RoboDK station: Estación_kuka_ibero.rdk

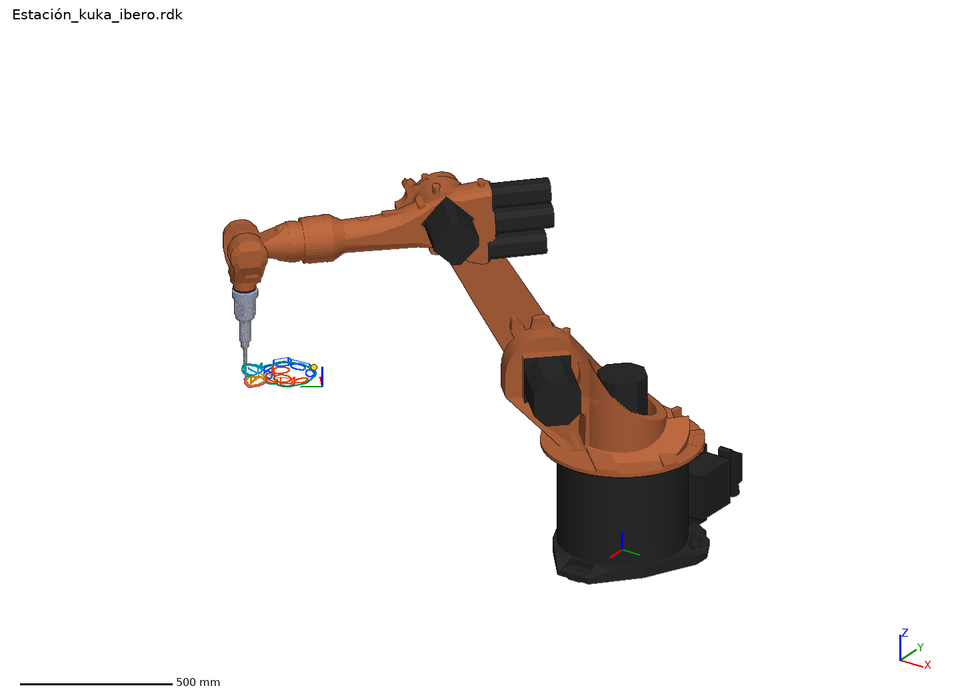
[picture v0: the station drawn from its stored meshes, robots at their saved joint values, targets as dots, program paths as lines]
Station Estación_kuka_ibero (saved by RoboDK 5.9.0). Poses are relative to the parent item; angles as X-Y-Z fixed-axis rotations.
  - frame KUKA KR 16 2 Base at (0, 0, 1020) mm, rotated rx 0 ry 0 rz -90 deg
    - robot KUKA KR 16 2: 6 axes, payload 16 kg, reach 1611 mm, repeatability 0.05 mm, weight 235 kg
        modified DH rows (alpha deg, a mm, theta deg, d mm): 0, 0, 0, 675; -90, 260, 0, 0; 0, 680, -90, 0; -90, -35, 0, 670; 90, 0, 0, 0; -90, 0, 180, 158
        joint limits [-185, -155, -130, -350, -130, -350] to [185, 35, 154, 350, 130, 350]; home [0, -90, 90, 0, 0, 0]; saved at [45.036, -60.88, 62.472, -0.86, 88.364, 45.057]
      - tool Plumon_ensamble, TCP at (4.25, 1.36, 301.29) mm, size 85.6 x 85.6 x 301.8 mm, geometry from Plumon_ensamble.IGS
  - object Celda_completa at (0, 0, 0) mm, size 7080 x 5029 x 2401 mm, geometry from Celda_completa.IGS
  - frame Frame 2 at (-643.65, -798.86, 1757.58) mm, rotated rx -0.03 ry 0.86 rz 129.82 deg
    - object RASPBERRY PI logo-0 at (0, 0, 0) mm
  - machining project P_in_1: rotZ(0) | rotX(0)*rotY(0) | rotz(0) | onStart | onPathStart | onApproach | onPoint | onRetract | onFinish | SetRPM(%1) | SetTool(%1) | Extruder(%1) | default | default | OutOnMov(%1) | OutOffMov(%1) | onPathFinish | M_RunCode(%1) | ag
  - program P_in_1 (855 instructions, listed below)
  - machining project P_in_2: rotZ(0) | rotX(0)*rotY(0) | rotz(0) | onStart | onPathStart | onApproach | onPoint | onRetract | onFinish | SetRPM(%1) | SetTool(%1) | Extruder(%1) | default | default | OutOnMov(%1) | OutOffMov(%1) | onPathFinish | M_RunCode(%1)
  - program P_in_2 (723 instructions, listed below)
  - machining project P_ou_1: rotZ(0) | rotX(0)*rotY(0) | rotz(0) | onStart | onPathStart | onApproach | onPoint | onRetract | onFinish | SetRPM(%1) | SetTool(%1) | Extruder(%1) | default | default | OutOnMov(%1) | OutOffMov(%1) | onPathFinish | M_RunCode(%1)
  - program P_ou_1 (860 instructions, listed below)
  - machining project P_ou_2: rotZ(0) | rotX(0)*rotY(0) | rotz(0) | onStart | onPathStart | onApproach | onPoint | onRetract | onFinish | SetRPM(%1) | SetTool(%1) | Extruder(%1) | default | default | OutOnMov(%1) | OutOffMov(%1) | onPathFinish | M_RunCode(%1)
  - program P_ou_2 (404 instructions, listed below)
  - machining project P_fl_1: rotZ(0) | rotX(0)*rotY(0) | rotz(0) | onStart | onPathStart | onApproach | onPoint | onRetract | onFinish | SetRPM(%1) | SetTool(%1) | Extruder(%1) | default | default | OutOnMov(%1) | OutOffMov(%1) | onPathFinish | M_RunCode(%1)
  - program P_fl_1 (618 instructions, listed below)
  - machining project P_fl_2: rotZ(0) | rotX(0)*rotY(0) | rotz(0) | onStart | onPathStart | onApproach | onPoint | onRetract | onFinish | SetRPM(%1) | SetTool(%1) | Extruder(%1) | default | default | OutOnMov(%1) | OutOffMov(%1) | onPathFinish | M_RunCode(%1)
  - program P_fl_2 (611 instructions, listed below)
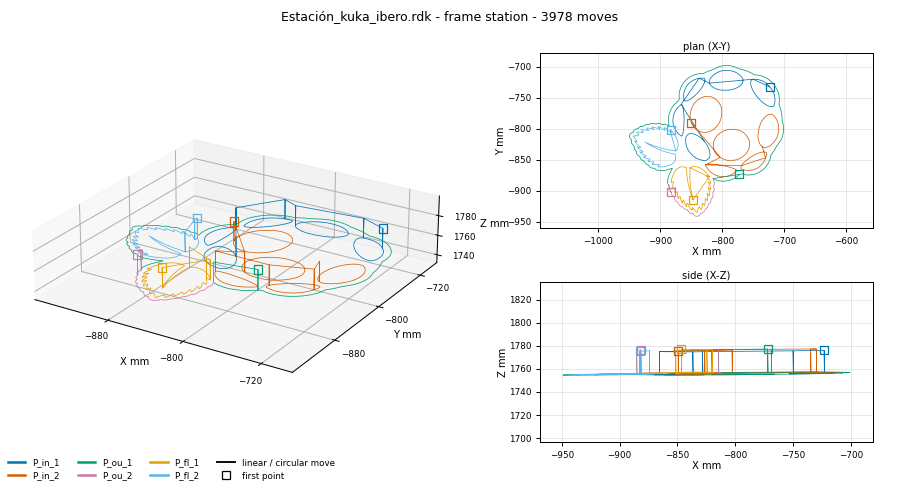
[picture p0: tool path of Estación_kuka_ibero.rdk in frame station, 3978 of 3978 moves have a stored position in this frame; points joined in program order, loops and branches not executed]

--- program P_in_1 (robot KUKA KR 16 2) ---
  Suave(1)
  Establecer velocidad (1000.0 mm/s)
  Est. Ref.: Frame 2
  Est. herr: Plumon_ensamble
  Mostrar Plumon_ensamble
  MoveJ 1 to (101.69, 18.24, 20) mm, rotated rx -180 ry 0 rz -39.83 deg; joints [44.906, -80.315, 88.498, -0.868, 81.773, 45.027]
  MoveL 2 to (101.69, 18.24, 20) mm, rotated rx -180 ry 0 rz -39.83 deg; joints [44.906, -80.315, 88.498, -0.868, 81.773, 45.027]
  MoveL 3 to (101.69, 18.24, 0) mm, rotated rx 180 ry 0 rz -39.83 deg; joints [44.889, -79.963, 89.829, -0.872, 80.089, 45.036]
  MoveL 4 to (101.69, 18.24, 0) mm, rotated rx 180 ry 0 rz -39.83 deg; joints [44.889, -79.963, 89.829, -0.872, 80.089, 45.036]
  Establecer velocidad (50.0 mm/s)
  MoveL 5 to (102.01, 18.23, 0) mm, rotated rx -180 ry 0 rz -39.83 deg; joints [44.907, -79.966, 89.833, -0.872, 80.088, 45.054]
  MoveL 6 to (102.33, 18.22, 0) mm, rotated rx -180 ry 0 rz -39.83 deg; joints [44.925, -79.969, 89.836, -0.872, 80.088, 45.071]
  MoveL 7 to (102.65, 18.22, 0) mm, rotated rx 180 ry 0 rz -39.83 deg; joints [44.942, -79.971, 89.84, -0.872, 80.087, 45.089]
  MoveL 8 to (102.97, 18.21, 0) mm, rotated rx 180 ry 0 rz -39.83 deg; joints [44.96, -79.974, 89.844, -0.872, 80.086, 45.106]
  MoveL 9 to (103.82, 18.21, 0) mm, rotated rx 180 ry 0 rz -39.83 deg; joints [45.007, -79.981, 89.853, -0.873, 80.085, 45.153]
  MoveL 10 to (104.66, 18.21, 0) mm, rotated rx 180 ry 0 rz -39.83 deg; joints [45.053, -79.986, 89.86, -0.873, 80.083, 45.2]
  MoveL 11 to (105.51, 18.24, 0) mm, rotated rx -180 ry 0 rz -39.83 deg; joints [45.1, -79.99, 89.866, -0.873, 80.082, 45.247]
  MoveL 12 to (106.35, 18.29, 0) mm, rotated rx 180 ry 0 rz -39.83 deg; joints [45.147, -79.991, 89.869, -0.873, 80.081, 45.294]
  MoveL 13 to (107.28, 18.4, 0) mm, rotated rx 180 ry 0 rz -39.83 deg; joints [45.199, -79.989, 89.867, -0.873, 80.081, 45.346]
  MoveL 14 to (108.21, 18.54, 0) mm, rotated rx 180 ry 0 rz -39.83 deg; joints [45.251, -79.984, 89.863, -0.873, 80.082, 45.398]
  MoveL 15 to (109.14, 18.7, 0) mm, rotated rx 180 ry 0 rz -39.83 deg; joints [45.303, -79.977, 89.855, -0.873, 80.083, 45.45]
  MoveL 16 to (110.07, 18.89, 0) mm, rotated rx 180 ry 0 rz -39.83 deg; joints [45.355, -79.968, 89.846, -0.873, 80.084, 45.502]
  MoveL 17 to (110.67, 19.01, 0) mm, rotated rx 180 ry 0 rz -39.83 deg; joints [45.389, -79.961, 89.839, -0.873, 80.085, 45.536]
  MoveL 18 to (111.27, 19.15, 0) mm, rotated rx -180 ry 0 rz -39.83 deg; joints [45.423, -79.954, 89.831, -0.873, 80.086, 45.57]
  MoveL 19 to (111.86, 19.3, 0) mm, rotated rx 180 ry 0 rz -39.83 deg; joints [45.456, -79.946, 89.822, -0.873, 80.087, 45.603]
  MoveL 20 to (112.45, 19.46, 0) mm, rotated rx 180 ry 0 rz -39.83 deg; joints [45.49, -79.936, 89.811, -0.873, 80.089, 45.636]
  MoveL 21 to (112.98, 19.63, 0) mm, rotated rx 180 ry 0 rz -39.83 deg; joints [45.52, -79.926, 89.8, -0.873, 80.09, 45.666]
  MoveL 22 to (113.5, 19.82, 0) mm, rotated rx -180 ry 0 rz -39.83 deg; joints [45.549, -79.914, 89.786, -0.873, 80.092, 45.696]
  MoveL 23 to (114.02, 20.01, 0) mm, rotated rx 180 ry 0 rz -39.83 deg; joints [45.579, -79.901, 89.772, -0.873, 80.094, 45.726]
  MoveL 24 to (114.54, 20.22, 0) mm, rotated rx -180 ry 0 rz -39.83 deg; joints [45.608, -79.888, 89.757, -0.873, 80.096, 45.755]
  MoveL 25 to (114.92, 20.37, 0) mm, rotated rx -180 ry 0 rz -39.83 deg; joints [45.63, -79.877, 89.745, -0.873, 80.098, 45.777]
  MoveL 26 to (115.3, 20.53, 0) mm, rotated rx 180 ry 0 rz -39.83 deg; joints [45.652, -79.867, 89.733, -0.873, 80.1, 45.799]
  MoveL 27 to (115.68, 20.69, 0) mm, rotated rx 180 ry 0 rz -39.83 deg; joints [45.674, -79.856, 89.721, -0.873, 80.102, 45.82]
  MoveL 28 to (116.05, 20.86, 0) mm, rotated rx 180 ry 0 rz -39.83 deg; joints [45.695, -79.844, 89.707, -0.873, 80.104, 45.842]
  MoveL 29 to (116.62, 21.14, 0) mm, rotated rx -180 ry 0 rz -39.83 deg; joints [45.728, -79.825, 89.686, -0.873, 80.107, 45.874]
  MoveL 30 to (117.19, 21.42, 0) mm, rotated rx -180 ry 0 rz -39.83 deg; joints [45.76, -79.805, 89.663, -0.873, 80.11, 45.907]
  MoveL 31 to (117.75, 21.72, 0) mm, rotated rx -180 ry 0 rz -39.83 deg; joints [45.792, -79.784, 89.638, -0.873, 80.114, 45.939]
  MoveL 32 to (118.3, 22.03, 0) mm, rotated rx -180 ry 0 rz -39.83 deg; joints [45.824, -79.762, 89.613, -0.873, 80.118, 45.97]
  MoveL 33 to (118.89, 22.38, 0) mm, rotated rx 180 ry 0 rz -39.83 deg; joints [45.858, -79.737, 89.584, -0.873, 80.122, 46.004]
  MoveL 34 to (119.47, 22.73, 0) mm, rotated rx -180 ry 0 rz -39.83 deg; joints [45.892, -79.712, 89.555, -0.873, 80.126, 46.038]
  MoveL 35 to (120.05, 23.09, 0) mm, rotated rx -180 ry 0 rz -39.83 deg; joints [45.925, -79.685, 89.525, -0.873, 80.131, 46.071]
  MoveL 36 to (120.62, 23.46, 0) mm, rotated rx 180 ry 0 rz -39.83 deg; joints [45.958, -79.658, 89.493, -0.873, 80.136, 46.104]
  MoveL 37 to (121.16, 23.83, 0) mm, rotated rx -180 ry 0 rz -39.83 deg; joints [45.989, -79.631, 89.462, -0.873, 80.141, 46.135]
  MoveL 38 to (121.69, 24.21, 0) mm, rotated rx 180 ry 0 rz -39.83 deg; joints [46.02, -79.603, 89.429, -0.873, 80.146, 46.166]
  MoveL 39 to (122.22, 24.59, 0) mm, rotated rx -180 ry 0 rz -39.83 deg; joints [46.05, -79.574, 89.396, -0.873, 80.151, 46.196]
  MoveL 40 to (122.73, 24.99, 0) mm, rotated rx 180 ry 0 rz -39.83 deg; joints [46.08, -79.545, 89.361, -0.873, 80.156, 46.226]
  MoveL 41 to (123.24, 25.41, 0) mm, rotated rx 180 ry 0 rz -39.83 deg; joints [46.11, -79.513, 89.325, -0.873, 80.162, 46.256]
  MoveL 42 to (123.74, 25.84, 0) mm, rotated rx 180 ry 0 rz -39.83 deg; joints [46.139, -79.481, 89.287, -0.873, 80.168, 46.285]
  MoveL 43 to (124.23, 26.28, 0) mm, rotated rx 180 ry 0 rz -39.83 deg; joints [46.168, -79.447, 89.247, -0.873, 80.174, 46.313]
  MoveL 44 to (124.7, 26.74, 0) mm, rotated rx -180 ry 0 rz -39.83 deg; joints [46.195, -79.412, 89.206, -0.873, 80.18, 46.341]
  MoveL 45 to (125.16, 27.22, 0) mm, rotated rx 180 ry 0 rz -39.83 deg; joints [46.223, -79.375, 89.163, -0.873, 80.187, 46.368]
  MoveL 46 to (125.61, 27.71, 0) mm, rotated rx 180 ry 0 rz -39.83 deg; joints [46.249, -79.337, 89.118, -0.873, 80.194, 46.394]
  MoveL 47 to (126.06, 28.2, 0) mm, rotated rx 180 ry 0 rz -39.83 deg; joints [46.276, -79.299, 89.074, -0.873, 80.201, 46.421]
  MoveL 48 to (126.51, 28.69, 0) mm, rotated rx 180 ry 0 rz -39.83 deg; joints [46.302, -79.262, 89.03, -0.873, 80.208, 46.448]
  MoveL 49 to (126.76, 28.95, 0) mm, rotated rx 180 ry 0 rz -39.83 deg; joints [46.317, -79.242, 89.006, -0.873, 80.212, 46.462]
  MoveL 50 to (127.01, 29.21, 0) mm, rotated rx 180 ry 0 rz -39.83 deg; joints [46.332, -79.222, 88.983, -0.873, 80.216, 46.477]
  MoveL 51 to (127.25, 29.47, 0) mm, rotated rx 180 ry 0 rz -39.83 deg; joints [46.346, -79.202, 88.959, -0.873, 80.22, 46.491]
  MoveL 52 to (127.48, 29.74, 0) mm, rotated rx -180 ry 0 rz -39.83 deg; joints [46.36, -79.18, 88.934, -0.873, 80.224, 46.504]
  MoveL 53 to (127.71, 30.06, 0) mm, rotated rx 180 ry 0 rz -39.83 deg; joints [46.373, -79.156, 88.905, -0.873, 80.228, 46.518]
  MoveL 54 to (127.92, 30.38, 0) mm, rotated rx -180 ry 0 rz -39.83 deg; joints [46.386, -79.131, 88.874, -0.873, 80.233, 46.531]
  MoveL 55 to (128.12, 30.71, 0) mm, rotated rx 180 ry 0 rz -39.83 deg; joints [46.398, -79.104, 88.843, -0.873, 80.238, 46.543]
  MoveL 56 to (128.32, 31.05, 0) mm, rotated rx 180 ry 0 rz -39.83 deg; joints [46.41, -79.077, 88.812, -0.873, 80.243, 46.555]
  Establecer velocidad (1000.0 mm/s)
  MoveL 57 to (128.32, 31.05, 0) mm, rotated rx 180 ry 0 rz -39.83 deg; joints [46.41, -79.077, 88.812, -0.873, 80.243, 46.555]
  MoveL 58 to (128.32, 31.05, 20) mm, rotated rx 180 ry 0 rz -39.83 deg; joints [46.427, -79.425, 87.481, -0.869, 81.922, 46.545]
  Establecer velocidad (1000.0 mm/s)
  MoveL 59 to (101.69, 18.24, 20) mm, rotated rx -180 ry 0 rz -39.83 deg; joints [44.906, -80.315, 88.498, -0.868, 81.773, 45.027]
  MoveL 60 to (101.69, 18.24, 0) mm, rotated rx 180 ry 0 rz -39.83 deg; joints [44.889, -79.963, 89.829, -0.872, 80.089, 45.036]
  MoveL 61 to (101.69, 18.24, 0) mm, rotated rx 180 ry 0 rz -39.83 deg; joints [44.889, -79.963, 89.829, -0.872, 80.089, 45.036]
  Establecer velocidad (50.0 mm/s)
  MoveL 62 to (101.37, 18.23, 0) mm, rotated rx -180 ry 0 rz -39.83 deg; joints [44.872, -79.961, 89.826, -0.872, 80.089, 45.018]
  MoveL 63 to (101.06, 18.22, 0) mm, rotated rx 180 ry 0 rz -39.83 deg; joints [44.854, -79.959, 89.824, -0.872, 80.09, 45.001]
  MoveL 64 to (100.74, 18.22, 0) mm, rotated rx 180 ry 0 rz -39.83 deg; joints [44.836, -79.957, 89.821, -0.872, 80.09, 44.983]
  MoveL 65 to (100.42, 18.21, 0) mm, rotated rx 180 ry 0 rz -39.83 deg; joints [44.819, -79.955, 89.818, -0.872, 80.091, 44.965]
  MoveL 66 to (99.57, 18.21, 0) mm, rotated rx -180 ry 0 rz -39.83 deg; joints [44.772, -79.95, 89.811, -0.872, 80.092, 44.918]
  MoveL 67 to (98.72, 18.21, 0) mm, rotated rx 180 ry 0 rz -39.83 deg; joints [44.725, -79.943, 89.801, -0.872, 80.094, 44.872]
  MoveL 68 to (97.88, 18.24, 0) mm, rotated rx 180 ry 0 rz -39.83 deg; joints [44.679, -79.935, 89.79, -0.872, 80.096, 44.825]
  MoveL 69 to (97.04, 18.29, 0) mm, rotated rx 180 ry 0 rz -39.83 deg; joints [44.633, -79.924, 89.776, -0.872, 80.098, 44.779]
  MoveL 70 to (96.1, 18.4, 0) mm, rotated rx 180 ry 0 rz -39.83 deg; joints [44.582, -79.908, 89.756, -0.872, 80.102, 44.728]
  MoveL 71 to (95.17, 18.54, 0) mm, rotated rx 180 ry 0 rz -39.83 deg; joints [44.531, -79.889, 89.733, -0.872, 80.105, 44.677]
  MoveL 72 to (94.25, 18.7, 0) mm, rotated rx 180 ry 0 rz -39.83 deg; joints [44.481, -79.868, 89.707, -0.872, 80.11, 44.627]
  MoveL 73 to (93.32, 18.89, 0) mm, rotated rx 180 ry 0 rz -39.83 deg; joints [44.431, -79.846, 89.679, -0.872, 80.114, 44.577]
  MoveL 74 to (92.72, 19.01, 0) mm, rotated rx -180 ry 0 rz -39.83 deg; joints [44.398, -79.831, 89.661, -0.872, 80.117, 44.544]
  MoveL 75 to (92.12, 19.15, 0) mm, rotated rx 180 ry 0 rz -39.83 deg; joints [44.366, -79.815, 89.641, -0.872, 80.121, 44.512]
  MoveL 76 to (91.53, 19.3, 0) mm, rotated rx 180 ry 0 rz -39.83 deg; joints [44.334, -79.798, 89.62, -0.872, 80.124, 44.48]
  MoveL 77 to (90.94, 19.46, 0) mm, rotated rx 180 ry 0 rz -39.83 deg; joints [44.303, -79.779, 89.598, -0.872, 80.128, 44.449]
  MoveL 78 to (90.41, 19.63, 0) mm, rotated rx 180 ry 0 rz -39.83 deg; joints [44.275, -79.761, 89.576, -0.872, 80.131, 44.42]
  MoveL 79 to (89.89, 19.82, 0) mm, rotated rx -180 ry 0 rz -39.83 deg; joints [44.247, -79.742, 89.552, -0.872, 80.135, 44.393]
  MoveL 80 to (89.37, 20.01, 0) mm, rotated rx 180 ry 0 rz -39.83 deg; joints [44.219, -79.722, 89.527, -0.872, 80.139, 44.365]
  MoveL 81 to (88.85, 20.22, 0) mm, rotated rx 180 ry 0 rz -39.83 deg; joints [44.192, -79.701, 89.502, -0.872, 80.143, 44.338]
  MoveL 82 to (88.47, 20.37, 0) mm, rotated rx 180 ry 0 rz -39.83 deg; joints [44.172, -79.685, 89.482, -0.872, 80.146, 44.318]
  MoveL 83 to (88.09, 20.53, 0) mm, rotated rx 180 ry 0 rz -39.83 deg; joints [44.152, -79.669, 89.463, -0.872, 80.15, 44.297]
  MoveL 84 to (87.71, 20.69, 0) mm, rotated rx 180 ry 0 rz -39.83 deg; joints [44.132, -79.652, 89.443, -0.872, 80.153, 44.278]
  MoveL 85 to (87.33, 20.86, 0) mm, rotated rx -180 ry 0 rz -39.83 deg; joints [44.112, -79.635, 89.422, -0.872, 80.156, 44.258]
  MoveL 86 to (86.76, 21.14, 0) mm, rotated rx 180 ry 0 rz -39.83 deg; joints [44.083, -79.608, 89.389, -0.871, 80.162, 44.228]
  MoveL 87 to (86.2, 21.42, 0) mm, rotated rx 180 ry 0 rz -39.83 deg; joints [44.053, -79.58, 89.355, -0.871, 80.167, 44.199]
  MoveL 88 to (85.64, 21.72, 0) mm, rotated rx 180 ry 0 rz -39.83 deg; joints [44.025, -79.55, 89.319, -0.871, 80.173, 44.17]
  MoveL 89 to (85.09, 22.03, 0) mm, rotated rx -180 ry 0 rz -39.83 deg; joints [43.996, -79.52, 89.283, -0.871, 80.179, 44.141]
  MoveL 90 to (84.5, 22.38, 0) mm, rotated rx 180 ry 0 rz -39.83 deg; joints [43.966, -79.487, 89.242, -0.871, 80.186, 44.111]
  MoveL 91 to (83.91, 22.73, 0) mm, rotated rx 180 ry 0 rz -39.83 deg; joints [43.936, -79.453, 89.201, -0.871, 80.192, 44.081]
  MoveL 92 to (83.34, 23.09, 0) mm, rotated rx 180 ry 0 rz -39.83 deg; joints [43.906, -79.419, 89.16, -0.871, 80.199, 44.051]
  MoveL 93 to (82.76, 23.46, 0) mm, rotated rx -180 ry 0 rz -39.83 deg; joints [43.877, -79.383, 89.117, -0.871, 80.206, 44.022]
  MoveL 94 to (82.23, 23.83, 0) mm, rotated rx 180 ry 0 rz -39.83 deg; joints [43.85, -79.349, 89.075, -0.871, 80.213, 43.994]
  MoveL 95 to (81.7, 24.21, 0) mm, rotated rx 180 ry 0 rz -39.83 deg; joints [43.823, -79.313, 89.032, -0.871, 80.22, 43.967]
  MoveL 96 to (81.17, 24.59, 0) mm, rotated rx 180 ry 0 rz -39.83 deg; joints [43.797, -79.277, 88.988, -0.871, 80.228, 43.941]
  MoveL 97 to (80.66, 24.99, 0) mm, rotated rx 180 ry 0 rz -39.83 deg; joints [43.771, -79.24, 88.943, -0.871, 80.235, 43.915]
  MoveL 98 to (80.15, 25.41, 0) mm, rotated rx 180 ry 0 rz -39.83 deg; joints [43.746, -79.201, 88.896, -0.871, 80.243, 43.89]
  MoveL 99 to (79.65, 25.84, 0) mm, rotated rx 180 ry 0 rz -39.83 deg; joints [43.721, -79.162, 88.848, -0.871, 80.251, 43.865]
  MoveL 100 to (79.16, 26.28, 0) mm, rotated rx 180 ry 0 rz -39.83 deg; joints [43.697, -79.121, 88.799, -0.871, 80.259, 43.841]
  MoveL 101 to (78.69, 26.74, 0) mm, rotated rx 180 ry 0 rz -39.83 deg; joints [43.675, -79.079, 88.748, -0.871, 80.267, 43.818]
  MoveL 102 to (78.23, 27.22, 0) mm, rotated rx -180 ry 0 rz -39.83 deg; joints [43.653, -79.036, 88.696, -0.871, 80.276, 43.796]
  MoveL 103 to (77.78, 27.71, 0) mm, rotated rx 180 ry 0 rz -39.83 deg; joints [43.631, -78.992, 88.642, -0.871, 80.285, 43.774]
  MoveL 104 to (77.33, 28.2, 0) mm, rotated rx -180 ry 0 rz -39.83 deg; joints [43.61, -78.947, 88.589, -0.871, 80.294, 43.753]
  MoveL 105 to (76.88, 28.69, 0) mm, rotated rx -180 ry 0 rz -39.83 deg; joints [43.588, -78.904, 88.535, -0.871, 80.303, 43.731]
  MoveL 106 to (76.63, 28.95, 0) mm, rotated rx -180 ry 0 rz -39.83 deg; joints [43.576, -78.88, 88.507, -0.871, 80.308, 43.719]
  MoveL 107 to (76.38, 29.21, 0) mm, rotated rx 180 ry 0 rz -39.83 deg; joints [43.564, -78.857, 88.479, -0.87, 80.313, 43.707]
  MoveL 108 to (76.14, 29.47, 0) mm, rotated rx 180 ry 0 rz -39.83 deg; joints [43.553, -78.833, 88.45, -0.87, 80.318, 43.695]
  MoveL 109 to (75.91, 29.74, 0) mm, rotated rx 180 ry 0 rz -39.83 deg; joints [43.542, -78.808, 88.42, -0.87, 80.323, 43.684]
  MoveL 110 to (75.68, 30.06, 0) mm, rotated rx 180 ry 0 rz -39.83 deg; joints [43.531, -78.781, 88.387, -0.87, 80.329, 43.674]
  MoveL 111 to (75.47, 30.38, 0) mm, rotated rx 180 ry 0 rz -39.83 deg; joints [43.522, -78.752, 88.352, -0.87, 80.335, 43.664]
  MoveL 112 to (75.27, 30.71, 0) mm, rotated rx -180 ry 0 rz -39.83 deg; joints [43.513, -78.723, 88.317, -0.87, 80.341, 43.656]
  MoveL 113 to (75.07, 31.05, 0) mm, rotated rx 180 ry 0 rz -39.83 deg; joints [43.505, -78.694, 88.281, -0.87, 80.347, 43.647]
  MoveL 114 to (75.07, 31.05, 0) mm, rotated rx 180 ry 0 rz -39.83 deg; joints [43.505, -78.694, 88.281, -0.87, 80.347, 43.647]
  MoveL 115 to (74.94, 31.32, 0) mm, rotated rx -180 ry 0 rz -39.83 deg; joints [43.5, -78.671, 88.253, -0.87, 80.351, 43.642]
  MoveL 116 to (74.82, 31.59, 0) mm, rotated rx 180 ry 0 rz -39.83 deg; joints [43.495, -78.648, 88.225, -0.87, 80.356, 43.637]
  MoveL 117 to (74.7, 31.86, 0) mm, rotated rx 180 ry 0 rz -39.83 deg; joints [43.49, -78.624, 88.197, -0.87, 80.361, 43.632]
  MoveL 118 to (74.6, 32.14, 0) mm, rotated rx 180 ry 0 rz -39.83 deg; joints [43.486, -78.601, 88.168, -0.87, 80.366, 43.628]
  MoveL 119 to (74.52, 32.35, 0) mm, rotated rx -180 ry 0 rz -39.83 deg; joints [43.483, -78.583, 88.147, -0.87, 80.37, 43.625]
  MoveL 120 to (74.46, 32.56, 0) mm, rotated rx 180 ry 0 rz -39.83 deg; joints [43.481, -78.565, 88.125, -0.87, 80.373, 43.623]
  MoveL 121 to (74.41, 32.78, 0) mm, rotated rx 180 ry 0 rz -39.83 deg; joints [43.48, -78.547, 88.103, -0.87, 80.377, 43.622]
  MoveL 122 to (74.37, 33, 0) mm, rotated rx 180 ry 0 rz -39.83 deg; joints [43.479, -78.528, 88.081, -0.87, 80.381, 43.621]
  MoveL 123 to (74.33, 33.36, 0) mm, rotated rx 180 ry 0 rz -39.83 deg; joints [43.479, -78.498, 88.045, -0.87, 80.387, 43.621]
  MoveL 124 to (74.32, 33.72, 0) mm, rotated rx 180 ry 0 rz -39.83 deg; joints [43.481, -78.469, 88.009, -0.87, 80.393, 43.622]
  MoveL 125 to (74.35, 34.09, 0) mm, rotated rx 180 ry 0 rz -39.83 deg; joints [43.485, -78.439, 87.973, -0.87, 80.4, 43.626]
  MoveL 126 to (74.42, 34.44, 0) mm, rotated rx 180 ry 0 rz -39.83 deg; joints [43.491, -78.411, 87.939, -0.87, 80.405, 43.632]
  MoveL 127 to (74.51, 34.76, 0) mm, rotated rx 180 ry 0 rz -39.83 deg; joints [43.498, -78.386, 87.909, -0.87, 80.411, 43.639]
  MoveL 128 to (74.63, 35.07, 0) mm, rotated rx 180 ry 0 rz -39.83 deg; joints [43.506, -78.362, 87.88, -0.87, 80.416, 43.647]
  MoveL 129 to (74.77, 35.37, 0) mm, rotated rx 180 ry 0 rz -39.83 deg; joints [43.516, -78.338, 87.852, -0.87, 80.42, 43.657]
  MoveL 130 to (74.94, 35.65, 0) mm, rotated rx 180 ry 0 rz -39.83 deg; joints [43.527, -78.316, 87.826, -0.87, 80.425, 43.668]
  MoveL 131 to (75.22, 36.07, 0) mm, rotated rx 180 ry 0 rz -39.83 deg; joints [43.544, -78.285, 87.788, -0.87, 80.432, 43.685]
  MoveL 132 to (75.53, 36.47, 0) mm, rotated rx 180 ry 0 rz -39.83 deg; joints [43.564, -78.255, 87.752, -0.87, 80.438, 43.705]
  MoveL 133 to (75.87, 36.85, 0) mm, rotated rx 180 ry 0 rz -39.83 deg; joints [43.584, -78.228, 87.719, -0.87, 80.443, 43.725]
  MoveL 134 to (76.23, 37.2, 0) mm, rotated rx -180 ry 0 rz -39.83 deg; joints [43.606, -78.202, 87.689, -0.87, 80.449, 43.747]
  MoveL 135 to (76.54, 37.48, 0) mm, rotated rx -180 ry 0 rz -39.83 deg; joints [43.624, -78.182, 87.665, -0.87, 80.453, 43.765]
  MoveL 136 to (76.85, 37.75, 0) mm, rotated rx 180 ry 0 rz -39.83 deg; joints [43.643, -78.163, 87.643, -0.87, 80.457, 43.784]
  MoveL 137 to (77.18, 38.01, 0) mm, rotated rx 180 ry 0 rz -39.83 deg; joints [43.662, -78.145, 87.621, -0.87, 80.46, 43.803]
  MoveL 138 to (77.51, 38.26, 0) mm, rotated rx 180 ry 0 rz -39.83 deg; joints [43.682, -78.127, 87.6, -0.87, 80.464, 43.822]
  MoveL 139 to (78.01, 38.62, 0) mm, rotated rx 180 ry 0 rz -39.83 deg; joints [43.711, -78.102, 87.57, -0.87, 80.469, 43.851]
  MoveL 140 to (78.52, 38.97, 0) mm, rotated rx 180 ry 0 rz -39.83 deg; joints [43.741, -78.078, 87.542, -0.87, 80.474, 43.881]
  MoveL 141 to (79.04, 39.3, 0) mm, rotated rx 180 ry 0 rz -39.83 deg; joints [43.77, -78.056, 87.515, -0.87, 80.478, 43.911]
  MoveL 142 to (79.57, 39.61, 0) mm, rotated rx 180 ry 0 rz -39.83 deg; joints [43.801, -78.035, 87.491, -0.87, 80.483, 43.941]
  MoveL 143 to (80.13, 39.9, 0) mm, rotated rx 180 ry 0 rz -39.83 deg; joints [43.833, -78.016, 87.469, -0.87, 80.486, 43.973]
  MoveL 144 to (80.71, 40.17, 0) mm, rotated rx 180 ry 0 rz -39.83 deg; joints [43.866, -77.999, 87.449, -0.87, 80.49, 44.006]
  MoveL 145 to (81.29, 40.42, 0) mm, rotated rx 180 ry 0 rz -39.83 deg; joints [43.899, -77.984, 87.431, -0.87, 80.493, 44.039]
  MoveL 146 to (81.88, 40.66, 0) mm, rotated rx -180 ry 0 rz -39.83 deg; joints [43.932, -77.969, 87.414, -0.87, 80.496, 44.072]
  MoveL 147 to (82.65, 40.97, 0) mm, rotated rx 180 ry 0 rz -39.83 deg; joints [43.975, -77.951, 87.392, -0.87, 80.499, 44.115]
  MoveL 148 to (83.42, 41.27, 0) mm, rotated rx -180 ry 0 rz -39.83 deg; joints [44.018, -77.933, 87.372, -0.871, 80.503, 44.158]
  MoveL 149 to (84.2, 41.55, 0) mm, rotated rx 180 ry 0 rz -39.83 deg; joints [44.062, -77.916, 87.353, -0.871, 80.506, 44.202]
  MoveL 150 to (84.98, 41.81, 0) mm, rotated rx 180 ry 0 rz -39.83 deg; joints [44.106, -77.902, 87.336, -0.871, 80.509, 44.246]
  MoveL 151 to (86.19, 42.17, 0) mm, rotated rx 180 ry 0 rz -39.83 deg; joints [44.173, -77.882, 87.314, -0.871, 80.512, 44.312]
  MoveL 152 to (87.4, 42.48, 0) mm, rotated rx 180 ry 0 rz -39.83 deg; joints [44.24, -77.867, 87.296, -0.871, 80.515, 44.38]
  MoveL 153 to (88.63, 42.76, 0) mm, rotated rx 180 ry 0 rz -39.83 deg; joints [44.307, -77.854, 87.283, -0.871, 80.517, 44.447]
  MoveL 154 to (89.86, 43.01, 0) mm, rotated rx -180 ry 0 rz -39.83 deg; joints [44.375, -77.844, 87.272, -0.871, 80.519, 44.515]
  MoveL 155 to (90.97, 43.22, 0) mm, rotated rx 180 ry 0 rz -39.83 deg; joints [44.436, -77.836, 87.263, -0.871, 80.52, 44.576]
  MoveL 156 to (92.08, 43.41, 0) mm, rotated rx 180 ry 0 rz -39.83 deg; joints [44.497, -77.829, 87.256, -0.871, 80.521, 44.637]
  MoveL 157 to (93.2, 43.58, 0) mm, rotated rx 180 ry 0 rz -39.83 deg; joints [44.558, -77.823, 87.251, -0.871, 80.522, 44.698]
  MoveL 158 to (94.31, 43.74, 0) mm, rotated rx 180 ry 0 rz -39.83 deg; joints [44.619, -77.819, 87.248, -0.871, 80.522, 44.759]
  MoveL 159 to (95.45, 43.87, 0) mm, rotated rx 180 ry 0 rz -39.83 deg; joints [44.68, -77.817, 87.246, -0.871, 80.522, 44.82]
  MoveL 160 to (96.62, 43.98, 0) mm, rotated rx 180 ry 0 rz -39.83 deg; joints [44.744, -77.817, 87.247, -0.871, 80.522, 44.884]
  MoveL 161 to (97.86, 44.07, 0) mm, rotated rx -180 ry 0 rz -39.83 deg; joints [44.811, -77.819, 87.252, -0.871, 80.52, 44.951]
  MoveL 162 to (99.2, 44.12, 0) mm, rotated rx 180 ry 0 rz -39.83 deg; joints [44.884, -77.825, 87.261, -0.871, 80.518, 45.024]
  MoveL 163 to (100.08, 44.13, 0) mm, rotated rx 180 ry 0 rz -39.83 deg; joints [44.932, -77.83, 87.269, -0.871, 80.517, 45.072]
  MoveL 164 to (100.89, 44.13, 0) mm, rotated rx 180 ry 0 rz -39.83 deg; joints [44.975, -77.836, 87.277, -0.871, 80.515, 45.115]
  MoveL 165 to (101.47, 44.13, 0) mm, rotated rx 180 ry 0 rz -39.83 deg; joints [45.006, -77.84, 87.283, -0.871, 80.514, 45.146]
  MoveL 166 to (101.69, 44.13, 0) mm, rotated rx 180 ry 0 rz -39.83 deg; joints [45.018, -77.842, 87.285, -0.871, 80.513, 45.159]
  MoveL 167 to (101.69, 44.13, 0) mm, rotated rx 180 ry 0 rz -39.83 deg; joints [45.018, -77.842, 87.285, -0.871, 80.513, 45.159]
  MoveL 168 to (101.92, 44.13, 0) mm, rotated rx 180 ry 0 rz -39.83 deg; joints [45.031, -77.843, 87.287, -0.871, 80.513, 45.171]
  MoveL 169 to (102.5, 44.13, 0) mm, rotated rx 180 ry 0 rz -39.83 deg; joints [45.062, -77.847, 87.293, -0.871, 80.512, 45.202]
  MoveL 170 to (103.3, 44.13, 0) mm, rotated rx -180 ry 0 rz -39.83 deg; joints [45.105, -77.853, 87.301, -0.871, 80.51, 45.245]
  MoveL 171 to (104.19, 44.12, 0) mm, rotated rx 180 ry 0 rz -39.83 deg; joints [45.153, -77.86, 87.311, -0.872, 80.508, 45.293]
  MoveL 172 to (105.53, 44.07, 0) mm, rotated rx -180 ry 0 rz -39.83 deg; joints [45.225, -77.874, 87.329, -0.872, 80.505, 45.365]
  MoveL 173 to (106.77, 43.98, 0) mm, rotated rx 180 ry 0 rz -39.83 deg; joints [45.292, -77.889, 87.349, -0.872, 80.501, 45.432]
  MoveL 174 to (107.94, 43.87, 0) mm, rotated rx 180 ry 0 rz -39.83 deg; joints [45.354, -77.906, 87.371, -0.872, 80.496, 45.495]
  MoveL 175 to (109.08, 43.74, 0) mm, rotated rx 180 ry 0 rz -39.83 deg; joints [45.415, -77.925, 87.395, -0.872, 80.492, 45.555]
  MoveL 176 to (110.19, 43.58, 0) mm, rotated rx 180 ry 0 rz -39.83 deg; joints [45.475, -77.945, 87.421, -0.872, 80.487, 45.615]
  MoveL 177 to (111.31, 43.41, 0) mm, rotated rx 180 ry 0 rz -39.83 deg; joints [45.534, -77.966, 87.449, -0.872, 80.482, 45.675]
  MoveL 178 to (112.42, 43.22, 0) mm, rotated rx 180 ry 0 rz -39.83 deg; joints [45.593, -77.989, 87.478, -0.872, 80.476, 45.734]
  MoveL 179 to (113.53, 43.01, 0) mm, rotated rx 180 ry 0 rz -39.83 deg; joints [45.652, -78.012, 87.508, -0.872, 80.471, 45.793]
  MoveL 180 to (114.76, 42.76, 0) mm, rotated rx -180 ry 0 rz -39.83 deg; joints [45.718, -78.04, 87.544, -0.872, 80.464, 45.859]
  MoveL 181 to (115.98, 42.48, 0) mm, rotated rx 180 ry 0 rz -39.83 deg; joints [45.783, -78.071, 87.582, -0.872, 80.457, 45.924]
  MoveL 182 to (117.2, 42.17, 0) mm, rotated rx 180 ry 0 rz -39.83 deg; joints [45.848, -78.104, 87.624, -0.872, 80.449, 45.989]
  MoveL 183 to (118.4, 41.81, 0) mm, rotated rx 180 ry 0 rz -39.83 deg; joints [45.911, -78.14, 87.669, -0.872, 80.441, 46.053]
  MoveL 184 to (119.19, 41.55, 0) mm, rotated rx -180 ry 0 rz -39.83 deg; joints [45.953, -78.166, 87.702, -0.872, 80.435, 46.094]
  MoveL 185 to (119.97, 41.27, 0) mm, rotated rx -180 ry 0 rz -39.83 deg; joints [45.994, -78.194, 87.737, -0.872, 80.428, 46.135]
  MoveL 186 to (120.74, 40.97, 0) mm, rotated rx -180 ry 0 rz -39.83 deg; joints [46.035, -78.223, 87.773, -0.872, 80.422, 46.176]
  MoveL 187 to (121.51, 40.66, 0) mm, rotated rx -180 ry 0 rz -39.83 deg; joints [46.075, -78.252, 87.81, -0.872, 80.415, 46.217]
  MoveL 188 to (122.1, 40.42, 0) mm, rotated rx 180 ry 0 rz -39.83 deg; joints [46.106, -78.275, 87.838, -0.872, 80.41, 46.248]
  MoveL 189 to (122.68, 40.17, 0) mm, rotated rx 180 ry 0 rz -39.83 deg; joints [46.137, -78.299, 87.868, -0.872, 80.405, 46.279]
  MoveL 190 to (123.26, 39.9, 0) mm, rotated rx 180 ry 0 rz -39.83 deg; joints [46.167, -78.325, 87.899, -0.872, 80.399, 46.309]
  MoveL 191 to (123.82, 39.61, 0) mm, rotated rx 180 ry 0 rz -39.83 deg; joints [46.196, -78.351, 87.932, -0.872, 80.393, 46.339]
  MoveL 192 to (124.35, 39.3, 0) mm, rotated rx 180 ry 0 rz -39.83 deg; joints [46.224, -78.38, 87.967, -0.872, 80.387, 46.366]
  MoveL 193 to (124.87, 38.97, 0) mm, rotated rx 180 ry 0 rz -39.83 deg; joints [46.251, -78.41, 88.004, -0.873, 80.381, 46.393]
  MoveL 194 to (125.38, 38.62, 0) mm, rotated rx -180 ry 0 rz -39.83 deg; joints [46.277, -78.441, 88.043, -0.873, 80.374, 46.42]
  MoveL 195 to (125.88, 38.26, 0) mm, rotated rx 180 ry 0 rz -39.83 deg; joints [46.303, -78.473, 88.083, -0.873, 80.367, 46.446]
  MoveL 196 to (126.21, 38.01, 0) mm, rotated rx 180 ry 0 rz -39.83 deg; joints [46.32, -78.496, 88.11, -0.873, 80.362, 46.463]
  MoveL 197 to (126.53, 37.75, 0) mm, rotated rx 180 ry 0 rz -39.83 deg; joints [46.337, -78.519, 88.138, -0.873, 80.357, 46.48]
  MoveL 198 to (126.85, 37.48, 0) mm, rotated rx 180 ry 0 rz -39.83 deg; joints [46.353, -78.542, 88.167, -0.873, 80.352, 46.496]
  MoveL 199 to (127.16, 37.2, 0) mm, rotated rx 180 ry 0 rz -39.83 deg; joints [46.369, -78.567, 88.197, -0.873, 80.347, 46.512]
  MoveL 200 to (127.52, 36.85, 0) mm, rotated rx 180 ry 0 rz -39.83 deg; joints [46.388, -78.598, 88.235, -0.873, 80.34, 46.531]
  MoveL 201 to (127.86, 36.47, 0) mm, rotated rx 180 ry 0 rz -39.83 deg; joints [46.405, -78.63, 88.274, -0.873, 80.333, 46.548]
  MoveL 202 to (128.17, 36.07, 0) mm, rotated rx 180 ry 0 rz -39.83 deg; joints [46.42, -78.664, 88.316, -0.873, 80.326, 46.564]
  MoveL 203 to (128.45, 35.65, 0) mm, rotated rx 180 ry 0 rz -39.83 deg; joints [46.434, -78.7, 88.359, -0.873, 80.319, 46.577]
  MoveL 204 to (128.62, 35.37, 0) mm, rotated rx 180 ry 0 rz -39.83 deg; joints [46.442, -78.725, 88.389, -0.873, 80.314, 46.585]
  MoveL 205 to (128.76, 35.07, 0) mm, rotated rx 180 ry 0 rz -39.83 deg; joints [46.449, -78.75, 88.42, -0.873, 80.309, 46.592]
  MoveL 206 to (128.88, 34.76, 0) mm, rotated rx 180 ry 0 rz -39.83 deg; joints [46.454, -78.776, 88.451, -0.873, 80.303, 46.598]
  MoveL 207 to (128.97, 34.44, 0) mm, rotated rx -180 ry 0 rz -39.83 deg; joints [46.458, -78.802, 88.483, -0.873, 80.298, 46.602]
  MoveL 208 to (129.04, 34.09, 0) mm, rotated rx 180 ry 0 rz -39.83 deg; joints [46.46, -78.832, 88.519, -0.873, 80.292, 46.604]
  MoveL 209 to (129.07, 33.72, 0) mm, rotated rx 180 ry 0 rz -39.83 deg; joints [46.461, -78.862, 88.554, -0.873, 80.286, 46.605]
  MoveL 210 to (129.06, 33.36, 0) mm, rotated rx 180 ry 0 rz -39.83 deg; joints [46.459, -78.892, 88.59, -0.873, 80.28, 46.603]
  MoveL 211 to (129.02, 33, 0) mm, rotated rx 180 ry 0 rz -39.83 deg; joints [46.456, -78.921, 88.626, -0.873, 80.274, 46.6]
  MoveL 212 to (128.98, 32.78, 0) mm, rotated rx 180 ry 0 rz -39.83 deg; joints [46.453, -78.939, 88.647, -0.873, 80.271, 46.597]
  MoveL 213 to (128.93, 32.56, 0) mm, rotated rx 180 ry 0 rz -39.83 deg; joints [46.449, -78.957, 88.668, -0.873, 80.267, 46.593]
  MoveL 214 to (128.86, 32.35, 0) mm, rotated rx -180 ry 0 rz -39.83 deg; joints [46.445, -78.974, 88.688, -0.873, 80.264, 46.589]
  MoveL 215 to (128.79, 32.14, 0) mm, rotated rx 180 ry 0 rz -39.83 deg; joints [46.44, -78.991, 88.708, -0.873, 80.26, 46.584]
  MoveL 216 to (128.69, 31.86, 0) mm, rotated rx 180 ry 0 rz -39.83 deg; joints [46.433, -79.013, 88.735, -0.873, 80.256, 46.578]
  MoveL 217 to (128.57, 31.59, 0) mm, rotated rx 180 ry 0 rz -39.83 deg; joints [46.426, -79.035, 88.761, -0.873, 80.252, 46.57]
  MoveL 218 to (128.44, 31.32, 0) mm, rotated rx 180 ry 0 rz -39.83 deg; joints [46.418, -79.056, 88.786, -0.873, 80.248, 46.562]
  MoveL 219 to (128.32, 31.05, 0) mm, rotated rx 180 ry 0 rz -39.83 deg; joints [46.41, -79.077, 88.812, -0.873, 80.243, 46.555]
  Establecer velocidad (1000.0 mm/s)
  MoveL 220 to (128.32, 31.05, 0) mm, rotated rx 180 ry 0 rz -39.83 deg; joints [46.41, -79.077, 88.812, -0.873, 80.243, 46.555]
  MoveL 221 to (128.32, 31.05, 20) mm, rotated rx 180 ry 0 rz -39.83 deg; joints [46.427, -79.425, 87.481, -0.869, 81.922, 46.545]
  Establecer velocidad (1000.0 mm/s)
  MoveL 222 to (168.4, 89.11, 20) mm, rotated rx -180 ry 0 rz -39.83 deg; joints [48.709, -74.756, 81.792, -0.867, 82.976, 48.812]
  MoveL 223 to (168.4, 89.11, 0) mm, rotated rx 180 ry 0 rz -39.83 deg; joints [48.694, -74.438, 83.125, -0.871, 81.324, 48.822]
  MoveL 224 to (168.4, 89.11, 0) mm, rotated rx 180 ry 0 rz -39.83 deg; joints [48.694, -74.438, 83.125, -0.871, 81.324, 48.822]
  Establecer velocidad (50.0 mm/s)
  MoveL 225 to (167.87, 89.26, 0) mm, rotated rx -180 ry 0 rz -39.83 deg; joints [48.666, -74.425, 83.108, -0.871, 81.328, 48.794]
  MoveL 226 to (167.33, 89.39, 0) mm, rotated rx -180 ry 0 rz -39.83 deg; joints [48.638, -74.412, 83.092, -0.871, 81.332, 48.766]
  MoveL 227 to (166.79, 89.51, 0) mm, rotated rx 180 ry 0 rz -39.83 deg; joints [48.61, -74.401, 83.077, -0.871, 81.335, 48.738]
  MoveL 228 to (166.25, 89.61, 0) mm, rotated rx -180 ry 0 rz -39.83 deg; joints [48.582, -74.392, 83.065, -0.871, 81.338, 48.71]
  MoveL 229 to (165.14, 89.71, 0) mm, rotated rx 180 ry 0 rz -39.83 deg; joints [48.524, -74.382, 83.05, -0.871, 81.341, 48.652]
  MoveL 230 to (164.01, 89.69, 0) mm, rotated rx 180 ry 0 rz -39.83 deg; joints [48.466, -74.381, 83.047, -0.871, 81.342, 48.594]
  MoveL 231 to (162.89, 89.57, 0) mm, rotated rx 180 ry 0 rz -39.83 deg; joints [48.407, -74.388, 83.055, -0.871, 81.341, 48.535]
  MoveL 232 to (161.78, 89.36, 0) mm, rotated rx 180 ry 0 rz -39.83 deg; joints [48.349, -74.403, 83.073, -0.871, 81.337, 48.477]
  MoveL 233 to (160.86, 89.13, 0) mm, rotated rx 180 ry 0 rz -39.83 deg; joints [48.301, -74.42, 83.093, -0.871, 81.333, 48.429]
  MoveL 234 to (159.97, 88.85, 0) mm, rotated rx -180 ry 0 rz -39.83 deg; joints [48.254, -74.44, 83.118, -0.871, 81.328, 48.382]
  MoveL 235 to (159.09, 88.54, 0) mm, rotated rx -180 ry 0 rz -39.83 deg; joints [48.207, -74.464, 83.147, -0.871, 81.322, 48.336]
  MoveL 236 to (158.21, 88.2, 0) mm, rotated rx 180 ry 0 rz -39.83 deg; joints [48.161, -74.49, 83.179, -0.871, 81.315, 48.29]
  MoveL 237 to (157.52, 87.91, 0) mm, rotated rx 180 ry 0 rz -39.83 deg; joints [48.125, -74.512, 83.206, -0.871, 81.309, 48.253]
  MoveL 238 to (156.84, 87.61, 0) mm, rotated rx 180 ry 0 rz -39.83 deg; joints [48.088, -74.535, 83.235, -0.871, 81.303, 48.217]
  MoveL 239 to (156.15, 87.29, 0) mm, rotated rx -180 ry 0 rz -39.83 deg; joints [48.052, -74.56, 83.265, -0.871, 81.297, 48.181]
  MoveL 240 to (155.48, 86.96, 0) mm, rotated rx -180 ry 0 rz -39.83 deg; joints [48.016, -74.585, 83.296, -0.871, 81.29, 48.145]
  MoveL 241 to (154.69, 86.56, 0) mm, rotated rx -180 ry 0 rz -39.83 deg; joints [47.975, -74.616, 83.335, -0.871, 81.282, 48.103]
  MoveL 242 to (153.92, 86.14, 0) mm, rotated rx 180 ry 0 rz -39.83 deg; joints [47.933, -74.648, 83.375, -0.871, 81.274, 48.062]
  MoveL 243 to (153.16, 85.69, 0) mm, rotated rx -180 ry 0 rz -39.83 deg; joints [47.893, -74.683, 83.418, -0.871, 81.265, 48.022]
  MoveL 244 to (152.41, 85.22, 0) mm, rotated rx 180 ry 0 rz -39.83 deg; joints [47.853, -74.719, 83.464, -0.871, 81.255, 47.982]
  MoveL 245 to (151.64, 84.68, 0) mm, rotated rx 180 ry 0 rz -39.83 deg; joints [47.811, -74.761, 83.516, -0.871, 81.244, 47.941]
  MoveL 246 to (150.88, 84.12, 0) mm, rotated rx 180 ry 0 rz -39.83 deg; joints [47.771, -74.806, 83.572, -0.871, 81.232, 47.9]
  MoveL 247 to (150.15, 83.52, 0) mm, rotated rx 180 ry 0 rz -39.83 deg; joints [47.731, -74.853, 83.63, -0.871, 81.22, 47.86]
  MoveL 248 to (149.43, 82.9, 0) mm, rotated rx -180 ry 0 rz -39.83 deg; joints [47.692, -74.901, 83.691, -0.871, 81.207, 47.822]
  MoveL 249 to (148.81, 82.34, 0) mm, rotated rx -180 ry 0 rz -39.83 deg; joints [47.658, -74.946, 83.746, -0.871, 81.196, 47.788]
  MoveL 250 to (148.21, 81.77, 0) mm, rotated rx 180 ry 0 rz -39.83 deg; joints [47.625, -74.991, 83.803, -0.871, 81.184, 47.755]
  MoveL 251 to (147.61, 81.18, 0) mm, rotated rx 180 ry 0 rz -39.83 deg; joints [47.593, -75.037, 83.861, -0.871, 81.172, 47.723]
  MoveL 252 to (147.03, 80.59, 0) mm, rotated rx -180 ry 0 rz -39.83 deg; joints [47.561, -75.084, 83.92, -0.871, 81.159, 47.691]
  MoveL 253 to (146.43, 79.96, 0) mm, rotated rx 180 ry 0 rz -39.83 deg; joints [47.528, -75.134, 83.982, -0.871, 81.146, 47.659]
  MoveL 254 to (145.85, 79.32, 0) mm, rotated rx 180 ry 0 rz -39.83 deg; joints [47.496, -75.185, 84.045, -0.871, 81.133, 47.627]
  MoveL 255 to (145.28, 78.67, 0) mm, rotated rx -180 ry 0 rz -39.83 deg; joints [47.464, -75.236, 84.109, -0.871, 81.12, 47.595]
  MoveL 256 to (144.71, 78.02, 0) mm, rotated rx -180 ry 0 rz -39.83 deg; joints [47.433, -75.288, 84.174, -0.871, 81.107, 47.564]
  MoveL 257 to (144.17, 77.38, 0) mm, rotated rx 180 ry 0 rz -39.83 deg; joints [47.403, -75.338, 84.237, -0.871, 81.094, 47.534]
  MoveL 258 to (143.63, 76.74, 0) mm, rotated rx 180 ry 0 rz -39.83 deg; joints [47.373, -75.389, 84.3, -0.871, 81.081, 47.504]
  MoveL 259 to (143.09, 76.1, 0) mm, rotated rx 180 ry 0 rz -39.83 deg; joints [47.343, -75.44, 84.364, -0.871, 81.068, 47.475]
  MoveL 260 to (142.55, 75.45, 0) mm, rotated rx 180 ry 0 rz -39.83 deg; joints [47.313, -75.491, 84.427, -0.871, 81.055, 47.445]
  MoveL 261 to (142.03, 74.83, 0) mm, rotated rx 180 ry 0 rz -39.83 deg; joints [47.284, -75.541, 84.489, -0.871, 81.042, 47.416]
  MoveL 262 to (141.52, 74.2, 0) mm, rotated rx 180 ry 0 rz -39.83 deg; joints [47.255, -75.591, 84.551, -0.871, 81.03, 47.388]
  MoveL 263 to (141.03, 73.55, 0) mm, rotated rx 180 ry 0 rz -39.83 deg; joints [47.227, -75.642, 84.615, -0.871, 81.017, 47.36]
  MoveL 264 to (140.57, 72.89, 0) mm, rotated rx -180 ry 0 rz -39.83 deg; joints [47.201, -75.695, 84.681, -0.871, 81.003, 47.334]
  MoveL 265 to (140.13, 72.18, 0) mm, rotated rx -180 ry 0 rz -39.83 deg; joints [47.176, -75.751, 84.751, -0.871, 80.989, 47.309]
  MoveL 266 to (139.71, 71.46, 0) mm, rotated rx -180 ry 0 rz -39.83 deg; joints [47.152, -75.809, 84.823, -0.871, 80.975, 47.285]
  MoveL 267 to (139.31, 70.72, 0) mm, rotated rx 180 ry 0 rz -39.83 deg; joints [47.129, -75.868, 84.896, -0.871, 80.96, 47.262]
  MoveL 268 to (138.91, 69.99, 0) mm, rotated rx -180 ry 0 rz -39.83 deg; joints [47.105, -75.927, 84.969, -0.871, 80.945, 47.239]
  MoveL 269 to (138.43, 69.15, 0) mm, rotated rx 180 ry 0 rz -39.83 deg; joints [47.077, -75.994, 85.053, -0.871, 80.929, 47.212]
  MoveL 270 to (137.94, 68.3, 0) mm, rotated rx 180 ry 0 rz -39.83 deg; joints [47.049, -76.062, 85.137, -0.871, 80.912, 47.183]
  MoveL 271 to (137.46, 67.46, 0) mm, rotated rx 180 ry 0 rz -39.83 deg; joints [47.021, -76.129, 85.22, -0.871, 80.895, 47.156]
  MoveL 272 to (137, 66.6, 0) mm, rotated rx 180 ry 0 rz -39.83 deg; joints [46.995, -76.198, 85.306, -0.872, 80.879, 47.13]
  MoveL 273 to (136.68, 65.93, 0) mm, rotated rx 180 ry 0 rz -39.83 deg; joints [46.976, -76.252, 85.372, -0.872, 80.866, 47.111]
  MoveL 274 to (136.38, 65.25, 0) mm, rotated rx 180 ry 0 rz -39.83 deg; joints [46.958, -76.306, 85.44, -0.872, 80.852, 47.093]
  MoveL 275 to (136.1, 64.56, 0) mm, rotated rx -180 ry 0 rz -39.83 deg; joints [46.941, -76.362, 85.508, -0.872, 80.839, 47.076]
  MoveL 276 to (135.84, 63.87, 0) mm, rotated rx -180 ry 0 rz -39.83 deg; joints [46.925, -76.418, 85.578, -0.872, 80.825, 47.061]
  MoveL 277 to (135.56, 63.05, 0) mm, rotated rx 180 ry 0 rz -39.83 deg; joints [46.908, -76.484, 85.659, -0.872, 80.809, 47.043]
  MoveL 278 to (135.31, 62.22, 0) mm, rotated rx 180 ry 0 rz -39.83 deg; joints [46.891, -76.551, 85.742, -0.872, 80.793, 47.027]
  MoveL 279 to (135.07, 61.39, 0) mm, rotated rx -180 ry 0 rz -39.83 deg; joints [46.876, -76.618, 85.825, -0.872, 80.777, 47.013]
  MoveL 280 to (134.85, 60.55, 0) mm, rotated rx 180 ry 0 rz -39.83 deg; joints [46.862, -76.686, 85.909, -0.872, 80.761, 46.998]
  MoveL 281 to (134.59, 59.49, 0) mm, rotated rx 180 ry 0 rz -39.83 deg; joints [46.845, -76.772, 86.015, -0.872, 80.741, 46.982]
  MoveL 282 to (134.37, 58.42, 0) mm, rotated rx 180 ry 0 rz -39.83 deg; joints [46.83, -76.859, 86.123, -0.872, 80.72, 46.967]
  MoveL 283 to (134.18, 57.34, 0) mm, rotated rx 180 ry 0 rz -39.83 deg; joints [46.816, -76.947, 86.231, -0.872, 80.7, 46.953]
  MoveL 284 to (134.02, 56.25, 0) mm, rotated rx 180 ry 0 rz -39.83 deg; joints [46.804, -77.036, 86.34, -0.872, 80.679, 46.942]
  MoveL 285 to (133.94, 55.53, 0) mm, rotated rx -180 ry 0 rz -39.83 deg; joints [46.798, -77.095, 86.413, -0.872, 80.666, 46.936]
  MoveL 286 to (133.89, 54.8, 0) mm, rotated rx 180 ry 0 rz -39.83 deg; joints [46.792, -77.154, 86.486, -0.872, 80.652, 46.931]
  MoveL 287 to (133.86, 54.08, 0) mm, rotated rx -180 ry 0 rz -39.83 deg; joints [46.788, -77.214, 86.559, -0.872, 80.638, 46.927]
  MoveL 288 to (133.86, 53.35, 0) mm, rotated rx 180 ry 0 rz -39.83 deg; joints [46.786, -77.273, 86.632, -0.872, 80.625, 46.925]
  MoveL 289 to (133.89, 52.63, 0) mm, rotated rx 180 ry 0 rz -39.83 deg; joints [46.786, -77.333, 86.705, -0.872, 80.611, 46.924]
  MoveL 290 to (133.95, 51.9, 0) mm, rotated rx 180 ry 0 rz -39.83 deg; joints [46.787, -77.393, 86.779, -0.872, 80.597, 46.926]
  MoveL 291 to (134.05, 51.18, 0) mm, rotated rx 180 ry 0 rz -39.83 deg; joints [46.79, -77.453, 86.853, -0.872, 80.584, 46.929]
  MoveL 292 to (134.19, 50.46, 0) mm, rotated rx -180 ry 0 rz -39.83 deg; joints [46.795, -77.513, 86.926, -0.872, 80.57, 46.934]
  MoveL 293 to (134.34, 49.79, 0) mm, rotated rx 180 ry 0 rz -39.83 deg; joints [46.801, -77.568, 86.993, -0.872, 80.558, 46.941]
  MoveL 294 to (134.52, 49.14, 0) mm, rotated rx 180 ry 0 rz -39.83 deg; joints [46.809, -77.622, 87.06, -0.872, 80.545, 46.949]
  MoveL 295 to (134.75, 48.51, 0) mm, rotated rx 180 ry 0 rz -39.83 deg; joints [46.819, -77.676, 87.126, -0.872, 80.534, 46.959]
  MoveL 296 to (135.02, 47.89, 0) mm, rotated rx -180 ry 0 rz -39.83 deg; joints [46.831, -77.727, 87.189, -0.872, 80.522, 46.972]
  MoveL 297 to (135.39, 47.2, 0) mm, rotated rx 180 ry 0 rz -39.83 deg; joints [46.849, -77.785, 87.261, -0.872, 80.509, 46.99]
  MoveL 298 to (135.82, 46.55, 0) mm, rotated rx -180 ry 0 rz -39.83 deg; joints [46.871, -77.841, 87.329, -0.872, 80.497, 47.011]
  MoveL 299 to (136.31, 45.92, 0) mm, rotated rx 180 ry 0 rz -39.83 deg; joints [46.895, -77.895, 87.395, -0.872, 80.485, 47.036]
  MoveL 300 to (136.84, 45.32, 0) mm, rotated rx 180 ry 0 rz -39.83 deg; joints [46.922, -77.946, 87.458, -0.873, 80.473, 47.063]
  MoveL 301 to (137.43, 44.72, 0) mm, rotated rx 180 ry 0 rz -39.83 deg; joints [46.952, -77.998, 87.523, -0.873, 80.462, 47.093]
  MoveL 302 to (138.07, 44.17, 0) mm, rotated rx 180 ry 0 rz -39.83 deg; joints [46.985, -78.047, 87.582, -0.873, 80.451, 47.126]
  MoveL 303 to (138.75, 43.7, 0) mm, rotated rx 180 ry 0 rz -39.83 deg; joints [47.021, -78.088, 87.633, -0.873, 80.442, 47.162]
  MoveL 304 to (139.49, 43.34, 0) mm, rotated rx 180 ry 0 rz -39.83 deg; joints [47.059, -78.121, 87.674, -0.873, 80.434, 47.201]
  MoveL 305 to (140.16, 43.13, 0) mm, rotated rx -180 ry 0 rz -39.83 deg; joints [47.095, -78.141, 87.699, -0.873, 80.43, 47.237]
  MoveL 306 to (140.86, 43.01, 0) mm, rotated rx -180 ry 0 rz -39.83 deg; joints [47.133, -78.154, 87.715, -0.873, 80.427, 47.275]
  MoveL 307 to (141.58, 42.94, 0) mm, rotated rx 180 ry 0 rz -39.83 deg; joints [47.172, -78.162, 87.726, -0.873, 80.425, 47.314]
  MoveL 308 to (142.31, 42.92, 0) mm, rotated rx -180 ry 0 rz -39.83 deg; joints [47.211, -78.166, 87.733, -0.873, 80.423, 47.353]
  MoveL 309 to (143.2, 42.93, 0) mm, rotated rx 180 ry 0 rz -39.83 deg; joints [47.26, -78.169, 87.737, -0.873, 80.422, 47.402]
  MoveL 310 to (144.1, 42.97, 0) mm, rotated rx 180 ry 0 rz -39.83 deg; joints [47.308, -78.17, 87.739, -0.873, 80.422, 47.45]
  MoveL 311 to (144.98, 43.02, 0) mm, rotated rx -180 ry 0 rz -39.83 deg; joints [47.356, -78.169, 87.739, -0.873, 80.421, 47.498]
  MoveL 312 to (145.87, 43.09, 0) mm, rotated rx 180 ry 0 rz -39.83 deg; joints [47.405, -78.166, 87.737, -0.873, 80.421, 47.547]
  MoveL 313 to (146.77, 43.17, 0) mm, rotated rx 180 ry 0 rz -39.83 deg; joints [47.454, -78.163, 87.735, -0.873, 80.422, 47.596]
  MoveL 314 to (147.66, 43.27, 0) mm, rotated rx 180 ry 0 rz -39.83 deg; joints [47.503, -78.158, 87.73, -0.873, 80.422, 47.644]
  MoveL 315 to (148.55, 43.41, 0) mm, rotated rx 180 ry 0 rz -39.83 deg; joints [47.551, -78.15, 87.721, -0.873, 80.424, 47.693]
  MoveL 316 to (149.43, 43.59, 0) mm, rotated rx -180 ry 0 rz -39.83 deg; joints [47.599, -78.138, 87.708, -0.873, 80.426, 47.741]
  MoveL 317 to (150.33, 43.83, 0) mm, rotated rx -180 ry 0 rz -39.83 deg; joints [47.649, -78.121, 87.689, -0.873, 80.429, 47.791]
  MoveL 318 to (151.22, 44.12, 0) mm, rotated rx -180 ry 0 rz -39.83 deg; joints [47.698, -78.101, 87.665, -0.873, 80.433, 47.84]
  MoveL 319 to (152.11, 44.43, 0) mm, rotated rx 180 ry 0 rz -39.83 deg; joints [47.747, -78.078, 87.638, -0.873, 80.437, 47.888]
  MoveL 320 to (152.99, 44.74, 0) mm, rotated rx 180 ry 0 rz -39.83 deg; joints [47.795, -78.055, 87.611, -0.873, 80.442, 47.937]
  MoveL 321 to (153.77, 45.01, 0) mm, rotated rx -180 ry 0 rz -39.83 deg; joints [47.838, -78.035, 87.588, -0.873, 80.446, 47.98]
  MoveL 322 to (154.54, 45.29, 0) mm, rotated rx 180 ry 0 rz -39.83 deg; joints [47.881, -78.015, 87.565, -0.873, 80.449, 48.022]
  MoveL 323 to (155.31, 45.58, 0) mm, rotated rx -180 ry 0 rz -39.83 deg; joints [47.923, -77.993, 87.54, -0.873, 80.454, 48.064]
  MoveL 324 to (156.06, 45.9, 0) mm, rotated rx 180 ry 0 rz -39.83 deg; joints [47.964, -77.969, 87.511, -0.873, 80.459, 48.105]
  MoveL 325 to (156.85, 46.31, 0) mm, rotated rx 180 ry 0 rz -39.83 deg; joints [48.008, -77.938, 87.475, -0.873, 80.465, 48.149]
  MoveL 326 to (157.62, 46.75, 0) mm, rotated rx -180 ry 0 rz -39.83 deg; joints [48.05, -77.903, 87.434, -0.873, 80.472, 48.192]
  MoveL 327 to (158.38, 47.23, 0) mm, rotated rx 180 ry 0 rz -39.83 deg; joints [48.092, -77.866, 87.389, -0.873, 80.48, 48.233]
  MoveL 328 to (159.13, 47.72, 0) mm, rotated rx -180 ry 0 rz -39.83 deg; joints [48.134, -77.828, 87.343, -0.873, 80.488, 48.275]
  MoveL 329 to (160.13, 48.41, 0) mm, rotated rx 180 ry 0 rz -39.83 deg; joints [48.189, -77.774, 87.279, -0.873, 80.499, 48.33]
  MoveL 330 to (161.12, 49.12, 0) mm, rotated rx -180 ry 0 rz -39.83 deg; joints [48.244, -77.718, 87.212, -0.873, 80.511, 48.385]
  MoveL 331 to (162.08, 49.85, 0) mm, rotated rx 180 ry 0 rz -39.83 deg; joints [48.297, -77.66, 87.143, -0.873, 80.523, 48.438]
  MoveL 332 to (163.02, 50.62, 0) mm, rotated rx 180 ry 0 rz -39.83 deg; joints [48.349, -77.599, 87.069, -0.872, 80.536, 48.49]
  MoveL 333 to (163.87, 51.38, 0) mm, rotated rx 180 ry 0 rz -39.83 deg; joints [48.396, -77.538, 86.996, -0.872, 80.549, 48.536]
  MoveL 334 to (164.69, 52.18, 0) mm, rotated rx -180 ry 0 rz -39.83 deg; joints [48.442, -77.475, 86.919, -0.872, 80.563, 48.582]
  MoveL 335 to (165.48, 53, 0) mm, rotated rx 180 ry 0 rz -39.83 deg; joints [48.486, -77.409, 86.84, -0.872, 80.578, 48.626]
  MoveL 336 to (166.25, 53.85, 0) mm, rotated rx 180 ry 0 rz -39.83 deg; joints [48.529, -77.341, 86.757, -0.872, 80.593, 48.668]
  MoveL 337 to (167.06, 54.79, 0) mm, rotated rx 180 ry 0 rz -39.83 deg; joints [48.574, -77.265, 86.666, -0.872, 80.61, 48.713]
  MoveL 338 to (167.85, 55.75, 0) mm, rotated rx -180 ry 0 rz -39.83 deg; joints [48.617, -77.188, 86.572, -0.872, 80.627, 48.756]
  MoveL 339 to (168.6, 56.73, 0) mm, rotated rx 180 ry 0 rz -39.83 deg; joints [48.659, -77.108, 86.475, -0.872, 80.645, 48.798]
  MoveL 340 to (169.32, 57.74, 0) mm, rotated rx 180 ry 0 rz -39.83 deg; joints [48.699, -77.027, 86.375, -0.872, 80.663, 48.837]
  MoveL 341 to (170.01, 58.81, 0) mm, rotated rx 180 ry 0 rz -39.83 deg; joints [48.738, -76.94, 86.269, -0.872, 80.683, 48.876]
  MoveL 342 to (170.67, 59.92, 0) mm, rotated rx -180 ry 0 rz -39.83 deg; joints [48.774, -76.85, 86.159, -0.872, 80.704, 48.912]
  MoveL 343 to (171.26, 61.05, 0) mm, rotated rx 180 ry 0 rz -39.83 deg; joints [48.808, -76.758, 86.046, -0.872, 80.726, 48.945]
  MoveL 344 to (171.8, 62.21, 0) mm, rotated rx 180 ry 0 rz -39.83 deg; joints [48.838, -76.663, 85.929, -0.872, 80.748, 48.975]
  MoveL 345 to (172.18, 63.13, 0) mm, rotated rx -180 ry 0 rz -39.83 deg; joints [48.859, -76.588, 85.837, -0.872, 80.766, 48.996]
  MoveL 346 to (172.52, 64.05, 0) mm, rotated rx -180 ry 0 rz -39.83 deg; joints [48.878, -76.512, 85.743, -0.872, 80.784, 49.015]
  MoveL 347 to (172.83, 64.99, 0) mm, rotated rx 180 ry 0 rz -39.83 deg; joints [48.896, -76.436, 85.649, -0.872, 80.802, 49.033]
  MoveL 348 to (173.13, 65.94, 0) mm, rotated rx 180 ry 0 rz -39.83 deg; joints [48.913, -76.358, 85.553, -0.872, 80.821, 49.049]
  MoveL 349 to (173.39, 66.82, 0) mm, rotated rx 180 ry 0 rz -39.83 deg; joints [48.928, -76.286, 85.463, -0.872, 80.838, 49.064]
  MoveL 350 to (173.63, 67.7, 0) mm, rotated rx 180 ry 0 rz -39.83 deg; joints [48.942, -76.213, 85.373, -0.872, 80.856, 49.077]
  MoveL 351 to (173.85, 68.6, 0) mm, rotated rx -180 ry 0 rz -39.83 deg; joints [48.954, -76.14, 85.282, -0.872, 80.874, 49.09]
  MoveL 352 to (174.04, 69.49, 0) mm, rotated rx 180 ry 0 rz -39.83 deg; joints [48.966, -76.066, 85.19, -0.871, 80.892, 49.1]
  MoveL 353 to (174.21, 70.5, 0) mm, rotated rx 180 ry 0 rz -39.83 deg; joints [48.976, -75.984, 85.087, -0.871, 80.913, 49.111]
  MoveL 354 to (174.35, 71.51, 0) mm, rotated rx 180 ry 0 rz -39.83 deg; joints [48.984, -75.901, 84.983, -0.871, 80.934, 49.119]
  MoveL 355 to (174.46, 72.53, 0) mm, rotated rx 180 ry 0 rz -39.83 deg; joints [48.991, -75.817, 84.878, -0.871, 80.955, 49.125]
  MoveL 356 to (174.54, 73.55, 0) mm, rotated rx 180 ry 0 rz -39.83 deg; joints [48.996, -75.733, 84.773, -0.871, 80.976, 49.13]
  MoveL 357 to (174.59, 74.65, 0) mm, rotated rx 180 ry 0 rz -39.83 deg; joints [49.001, -75.642, 84.66, -0.871, 80.999, 49.134]
  MoveL 358 to (174.61, 75.75, 0) mm, rotated rx 180 ry 0 rz -39.83 deg; joints [49.003, -75.552, 84.546, -0.871, 81.022, 49.136]
  MoveL 359 to (174.6, 76.84, 0) mm, rotated rx 180 ry 0 rz -39.83 deg; joints [49.003, -75.461, 84.432, -0.871, 81.046, 49.136]
  MoveL 360 to (174.54, 77.94, 0) mm, rotated rx 180 ry 0 rz -39.83 deg; joints [49.001, -75.371, 84.318, -0.871, 81.069, 49.133]
  MoveL 361 to (174.44, 78.85, 0) mm, rotated rx 180 ry 0 rz -39.83 deg; joints [48.997, -75.295, 84.222, -0.871, 81.089, 49.129]
  MoveL 362 to (174.32, 79.77, 0) mm, rotated rx 180 ry 0 rz -39.83 deg; joints [48.992, -75.22, 84.126, -0.871, 81.109, 49.123]
  MoveL 363 to (174.15, 80.68, 0) mm, rotated rx -180 ry 0 rz -39.83 deg; joints [48.984, -75.144, 84.031, -0.871, 81.129, 49.115]
  MoveL 364 to (173.96, 81.58, 0) mm, rotated rx -180 ry 0 rz -39.83 deg; joints [48.975, -75.069, 83.936, -0.871, 81.149, 49.106]
  MoveL 365 to (173.72, 82.48, 0) mm, rotated rx 180 ry 0 rz -39.83 deg; joints [48.963, -74.995, 83.841, -0.871, 81.169, 49.094]
  MoveL 366 to (173.44, 83.36, 0) mm, rotated rx 180 ry 0 rz -39.83 deg; joints [48.95, -74.921, 83.748, -0.871, 81.189, 49.08]
  MoveL 367 to (173.11, 84.22, 0) mm, rotated rx 180 ry 0 rz -39.83 deg; joints [48.933, -74.85, 83.656, -0.871, 81.209, 49.063]
  MoveL 368 to (172.71, 85.06, 0) mm, rotated rx 180 ry 0 rz -39.83 deg; joints [48.913, -74.78, 83.568, -0.871, 81.228, 49.043]
  MoveL 369 to (172.46, 85.51, 0) mm, rotated rx 180 ry 0 rz -39.83 deg; joints [48.901, -74.742, 83.519, -0.871, 81.238, 49.03]
  MoveL 370 to (172.18, 85.95, 0) mm, rotated rx 180 ry 0 rz -39.83 deg; joints [48.887, -74.706, 83.472, -0.871, 81.248, 49.016]
  MoveL 371 to (171.88, 86.38, 0) mm, rotated rx 180 ry 0 rz -39.83 deg; joints [48.871, -74.67, 83.426, -0.871, 81.258, 49.001]
  MoveL 372 to (171.55, 86.79, 0) mm, rotated rx 180 ry 0 rz -39.83 deg; joints [48.855, -74.635, 83.381, -0.871, 81.268, 48.984]
  MoveL 373 to (171.14, 87.26, 0) mm, rotated rx 180 ry 0 rz -39.83 deg; joints [48.834, -74.596, 83.33, -0.871, 81.279, 48.963]
  MoveL 374 to (170.71, 87.7, 0) mm, rotated rx -180 ry 0 rz -39.83 deg; joints [48.812, -74.559, 83.283, -0.871, 81.289, 48.941]
  MoveL 375 to (170.23, 88.1, 0) mm, rotated rx 180 ry 0 rz -39.83 deg; joints [48.788, -74.525, 83.239, -0.871, 81.299, 48.916]
  MoveL 376 to (169.73, 88.45, 0) mm, rotated rx 180 ry 0 rz -39.83 deg; joints [48.762, -74.495, 83.2, -0.871, 81.307, 48.89]
  MoveL 377 to (169.41, 88.63, 0) mm, rotated rx 180 ry 0 rz -39.83 deg; joints [48.745, -74.479, 83.18, -0.871, 81.312, 48.874]
  MoveL 378 to (169.08, 88.8, 0) mm, rotated rx 180 ry 0 rz -39.83 deg; joints [48.728, -74.465, 83.161, -0.871, 81.316, 48.857]
  MoveL 379 to (168.74, 88.96, 0) mm, rotated rx 180 ry 0 rz -39.83 deg; joints [48.711, -74.451, 83.143, -0.871, 81.32, 48.839]
  MoveL 380 to (168.4, 89.11, 0) mm, rotated rx 180 ry 0 rz -39.83 deg; joints [48.694, -74.438, 83.125, -0.871, 81.324, 48.822]
  Establecer velocidad (1000.0 mm/s)
  MoveL 381 to (168.4, 89.11, 0) mm, rotated rx 180 ry 0 rz -39.83 deg; joints [48.694, -74.438, 83.125, -0.871, 81.324, 48.822]
  MoveL 382 to (168.4, 89.11, 20) mm, rotated rx -180 ry 0 rz -39.83 deg; joints [48.709, -74.756, 81.792, -0.867, 82.976, 48.812]
  Establecer velocidad (1000.0 mm/s)
  MoveL 383 to (185.15, 96.72, 20) mm, rotated rx 180 ry 0 rz -39.83 deg; joints [49.586, -74.143, 81.032, -0.867, 83.136, 49.687]
  MoveL 384 to (185.15, 96.72, 0) mm, rotated rx 180 ry 0 rz -39.83 deg; joints [49.571, -73.829, 82.367, -0.87, 81.487, 49.696]
  MoveL 385 to (185.15, 96.72, 0) mm, rotated rx 180 ry 0 rz -39.83 deg; joints [49.571, -73.829, 82.367, -0.87, 81.487, 49.696]
  Establecer velocidad (50.0 mm/s)
  MoveL 386 to (185.68, 97.63, 0) mm, rotated rx 180 ry 0 rz -39.83 deg; joints [49.598, -73.754, 82.271, -0.87, 81.508, 49.724]
  MoveL 387 to (186.19, 98.54, 0) mm, rotated rx -180 ry 0 rz -39.83 deg; joints [49.625, -73.679, 82.175, -0.87, 81.53, 49.75]
  MoveL 388 to (186.68, 99.46, 0) mm, rotated rx 180 ry 0 rz -39.83 deg; joints [49.651, -73.603, 82.077, -0.87, 81.552, 49.776]
  MoveL 389 to (187.14, 100.4, 0) mm, rotated rx 180 ry 0 rz -39.83 deg; joints [49.675, -73.525, 81.978, -0.87, 81.574, 49.799]
  MoveL 390 to (187.65, 101.6, 0) mm, rotated rx -180 ry 0 rz -39.83 deg; joints [49.702, -73.426, 81.85, -0.87, 81.603, 49.826]
  MoveL 391 to (188.09, 102.83, 0) mm, rotated rx 180 ry 0 rz -39.83 deg; joints [49.725, -73.324, 81.718, -0.869, 81.633, 49.849]
  MoveL 392 to (188.47, 104.08, 0) mm, rotated rx 180 ry 0 rz -39.83 deg; joints [49.745, -73.22, 81.584, -0.869, 81.663, 49.868]
  MoveL 393 to (188.79, 105.35, 0) mm, rotated rx -180 ry 0 rz -39.83 deg; joints [49.762, -73.115, 81.448, -0.869, 81.695, 49.885]
  MoveL 394 to (189.01, 106.5, 0) mm, rotated rx -180 ry 0 rz -39.83 deg; joints [49.774, -73.02, 81.324, -0.869, 81.723, 49.896]
  MoveL 395 to (189.19, 107.66, 0) mm, rotated rx 180 ry 0 rz -39.83 deg; joints [49.784, -72.924, 81.2, -0.869, 81.752, 49.905]
  MoveL 396 to (189.34, 108.82, 0) mm, rotated rx 180 ry 0 rz -39.83 deg; joints [49.791, -72.827, 81.074, -0.869, 81.781, 49.913]
  MoveL 397 to (189.45, 109.99, 0) mm, rotated rx 180 ry 0 rz -39.83 deg; joints [49.797, -72.73, 80.947, -0.869, 81.811, 49.918]
  MoveL 398 to (189.57, 111.89, 0) mm, rotated rx 180 ry 0 rz -39.83 deg; joints [49.804, -72.572, 80.741, -0.869, 81.86, 49.924]
  MoveL 399 to (189.59, 113.79, 0) mm, rotated rx -180 ry 0 rz -39.83 deg; joints [49.806, -72.414, 80.534, -0.869, 81.909, 49.925]
  MoveL 400 to (189.48, 115.68, 0) mm, rotated rx 180 ry 0 rz -39.83 deg; joints [49.801, -72.257, 80.327, -0.869, 81.958, 49.92]
  MoveL 401 to (189.21, 117.54, 0) mm, rotated rx 180 ry 0 rz -39.83 deg; joints [49.788, -72.102, 80.123, -0.869, 82.007, 49.906]
  MoveL 402 to (188.88, 118.94, 0) mm, rotated rx 180 ry 0 rz -39.83 deg; joints [49.771, -71.985, 79.969, -0.869, 82.044, 49.889]
  MoveL 403 to (188.45, 120.31, 0) mm, rotated rx 180 ry 0 rz -39.83 deg; joints [49.75, -71.87, 79.817, -0.869, 82.081, 49.867]
  MoveL 404 to (187.96, 121.67, 0) mm, rotated rx -180 ry 0 rz -39.83 deg; joints [49.726, -71.757, 79.666, -0.868, 82.118, 49.842]
  MoveL 405 to (187.42, 123.01, 0) mm, rotated rx -180 ry 0 rz -39.83 deg; joints [49.699, -71.645, 79.517, -0.868, 82.154, 49.815]
  MoveL 406 to (186.8, 124.45, 0) mm, rotated rx 180 ry 0 rz -39.83 deg; joints [49.669, -71.524, 79.357, -0.868, 82.194, 49.784]
  MoveL 407 to (186.14, 125.86, 0) mm, rotated rx 180 ry 0 rz -39.83 deg; joints [49.636, -71.406, 79.199, -0.868, 82.233, 49.75]
  MoveL 408 to (185.43, 127.24, 0) mm, rotated rx 180 ry 0 rz -39.83 deg; joints [49.601, -71.29, 79.044, -0.868, 82.271, 49.714]
  MoveL 409 to (184.63, 128.58, 0) mm, rotated rx 180 ry 0 rz -39.83 deg; joints [49.561, -71.178, 78.894, -0.868, 82.309, 49.674]
  MoveL 410 to (183.36, 130.36, 0) mm, rotated rx 180 ry 0 rz -39.83 deg; joints [49.498, -71.028, 78.692, -0.868, 82.36, 49.611]
  MoveL 411 to (181.92, 132.02, 0) mm, rotated rx -180 ry 0 rz -39.83 deg; joints [49.427, -70.888, 78.503, -0.868, 82.408, 49.539]
  MoveL 412 to (180.34, 133.56, 0) mm, rotated rx 180 ry 0 rz -39.83 deg; joints [49.349, -70.758, 78.327, -0.868, 82.453, 49.46]
  MoveL 413 to (178.65, 134.96, 0) mm, rotated rx -180 ry 0 rz -39.83 deg; joints [49.265, -70.638, 78.164, -0.868, 82.494, 49.376]
  MoveL 414 to (177.58, 135.74, 0) mm, rotated rx -180 ry 0 rz -39.83 deg; joints [49.213, -70.572, 78.073, -0.868, 82.518, 49.323]
  MoveL 415 to (176.5, 136.49, 0) mm, rotated rx 180 ry 0 rz -39.83 deg; joints [49.159, -70.508, 77.986, -0.868, 82.54, 49.269]
  MoveL 416 to (175.39, 137.2, 0) mm, rotated rx -180 ry 0 rz -39.83 deg; joints [49.105, -70.446, 77.902, -0.868, 82.562, 49.214]
  MoveL 417 to (174.28, 137.91, 0) mm, rotated rx 180 ry 0 rz -39.83 deg; joints [49.05, -70.385, 77.819, -0.868, 82.583, 49.159]
  MoveL 418 to (174.28, 137.91, 0) mm, rotated rx 180 ry 0 rz -39.83 deg; joints [49.05, -70.385, 77.819, -0.868, 82.583, 49.159]
  MoveL 419 to (174.1, 137.97, 0) mm, rotated rx 180 ry 0 rz -39.83 deg; joints [49.041, -70.38, 77.812, -0.868, 82.585, 49.15]
  MoveL 420 to (173.92, 138.02, 0) mm, rotated rx 180 ry 0 rz -39.83 deg; joints [49.032, -70.376, 77.805, -0.868, 82.587, 49.141]
  MoveL 421 to (173.74, 138.06, 0) mm, rotated rx 180 ry 0 rz -39.83 deg; joints [49.023, -70.372, 77.8, -0.868, 82.588, 49.132]
  MoveL 422 to (173.55, 138.09, 0) mm, rotated rx -180 ry 0 rz -39.83 deg; joints [49.014, -70.369, 77.796, -0.868, 82.589, 49.122]
  MoveL 423 to (173.31, 138.11, 0) mm, rotated rx -180 ry 0 rz -39.83 deg; joints [49.002, -70.367, 77.793, -0.868, 82.59, 49.11]
  MoveL 424 to (173.07, 138.1, 0) mm, rotated rx 180 ry 0 rz -39.83 deg; joints [48.99, -70.368, 77.794, -0.868, 82.59, 49.098]
  MoveL 425 to (172.83, 138.06, 0) mm, rotated rx 180 ry 0 rz -39.83 deg; joints [48.978, -70.371, 77.798, -0.868, 82.589, 49.086]
  MoveL 426 to (172.6, 137.99, 0) mm, rotated rx -180 ry 0 rz -39.83 deg; joints [48.966, -70.376, 77.804, -0.868, 82.587, 49.075]
  MoveL 427 to (172.36, 137.89, 0) mm, rotated rx 180 ry 0 rz -39.83 deg; joints [48.954, -70.384, 77.815, -0.868, 82.585, 49.063]
  MoveL 428 to (172.14, 137.76, 0) mm, rotated rx 180 ry 0 rz -39.83 deg; joints [48.943, -70.394, 77.828, -0.868, 82.581, 49.052]
  MoveL 429 to (171.92, 137.62, 0) mm, rotated rx 180 ry 0 rz -39.83 deg; joints [48.932, -70.406, 77.844, -0.868, 82.577, 49.041]
  MoveL 430 to (171.72, 137.46, 0) mm, rotated rx 180 ry 0 rz -39.83 deg; joints [48.922, -70.42, 77.862, -0.868, 82.573, 49.031]
  MoveL 431 to (171.43, 137.2, 0) mm, rotated rx -180 ry 0 rz -39.83 deg; joints [48.907, -70.441, 77.89, -0.868, 82.566, 49.016]
  MoveL 432 to (171.16, 136.91, 0) mm, rotated rx 180 ry 0 rz -39.83 deg; joints [48.893, -70.464, 77.921, -0.868, 82.558, 49.003]
  MoveL 433 to (170.92, 136.61, 0) mm, rotated rx -180 ry 0 rz -39.83 deg; joints [48.881, -70.489, 77.954, -0.868, 82.55, 48.99]
  MoveL 434 to (170.7, 136.3, 0) mm, rotated rx -180 ry 0 rz -39.83 deg; joints [48.869, -70.515, 77.989, -0.868, 82.541, 48.979]
  MoveL 435 to (170.48, 135.94, 0) mm, rotated rx 180 ry 0 rz -39.83 deg; joints [48.858, -70.545, 78.029, -0.868, 82.531, 48.968]
  MoveL 436 to (170.29, 135.56, 0) mm, rotated rx 180 ry 0 rz -39.83 deg; joints [48.848, -70.576, 78.07, -0.868, 82.52, 48.958]
  MoveL 437 to (170.11, 135.18, 0) mm, rotated rx 180 ry 0 rz -39.83 deg; joints [48.838, -70.608, 78.112, -0.868, 82.509, 48.948]
  MoveL 438 to (169.93, 134.79, 0) mm, rotated rx -180 ry 0 rz -39.83 deg; joints [48.829, -70.64, 78.155, -0.868, 82.498, 48.94]
  MoveL 439 to (169.93, 134.79, 0) mm, rotated rx -180 ry 0 rz -39.83 deg; joints [48.829, -70.64, 78.155, -0.868, 82.498, 48.94]
  MoveL 440 to (169.69, 134.14, 0) mm, rotated rx -180 ry 0 rz -39.83 deg; joints [48.816, -70.694, 78.228, -0.868, 82.48, 48.927]
  MoveL 441 to (169.45, 133.48, 0) mm, rotated rx -180 ry 0 rz -39.83 deg; joints [48.803, -70.749, 78.301, -0.868, 82.461, 48.914]
  MoveL 442 to (169.22, 132.82, 0) mm, rotated rx -180 ry 0 rz -39.83 deg; joints [48.791, -70.804, 78.374, -0.868, 82.443, 48.902]
  MoveL 443 to (169.02, 132.15, 0) mm, rotated rx 180 ry 0 rz -39.83 deg; joints [48.781, -70.86, 78.448, -0.868, 82.424, 48.892]
  MoveL 444 to (168.86, 131.49, 0) mm, rotated rx 180 ry 0 rz -39.83 deg; joints [48.772, -70.914, 78.521, -0.868, 82.406, 48.883]
  MoveL 445 to (168.72, 130.83, 0) mm, rotated rx -180 ry 0 rz -39.83 deg; joints [48.764, -70.97, 78.595, -0.868, 82.387, 48.876]
  MoveL 446 to (168.61, 130.16, 0) mm, rotated rx 180 ry 0 rz -39.83 deg; joints [48.757, -71.026, 78.67, -0.868, 82.369, 48.87]
  MoveL 447 to (168.52, 129.48, 0) mm, rotated rx 180 ry 0 rz -39.83 deg; joints [48.752, -71.082, 78.745, -0.868, 82.35, 48.865]
  MoveL 448 to (168.47, 128.87, 0) mm, rotated rx -180 ry 0 rz -39.83 deg; joints [48.748, -71.134, 78.813, -0.868, 82.333, 48.861]
  MoveL 449 to (168.42, 128.25, 0) mm, rotated rx 180 ry 0 rz -39.83 deg; joints [48.746, -71.185, 78.882, -0.868, 82.316, 48.859]
  MoveL 450 to (168.39, 127.63, 0) mm, rotated rx -180 ry 0 rz -39.83 deg; joints [48.743, -71.237, 78.95, -0.868, 82.299, 48.856]
  MoveL 451 to (168.37, 127.01, 0) mm, rotated rx -180 ry 0 rz -39.83 deg; joints [48.741, -71.288, 79.019, -0.868, 82.281, 48.855]
  MoveL 452 to (168.35, 126.2, 0) mm, rotated rx 180 ry 0 rz -39.83 deg; joints [48.74, -71.357, 79.11, -0.868, 82.259, 48.853]
  MoveL 453 to (168.35, 125.38, 0) mm, rotated rx -180 ry 0 rz -39.83 deg; joints [48.738, -71.425, 79.201, -0.869, 82.236, 48.852]
  MoveL 454 to (168.34, 124.56, 0) mm, rotated rx 180 ry 0 rz -39.83 deg; joints [48.737, -71.493, 79.291, -0.869, 82.214, 48.851]
  MoveL 455 to (168.34, 123.74, 0) mm, rotated rx 180 ry 0 rz -39.83 deg; joints [48.736, -71.561, 79.382, -0.869, 82.192, 48.851]
  MoveL 456 to (168.34, 122.71, 0) mm, rotated rx 180 ry 0 rz -39.83 deg; joints [48.734, -71.647, 79.496, -0.869, 82.164, 48.85]
  MoveL 457 to (168.34, 121.68, 0) mm, rotated rx 180 ry 0 rz -39.83 deg; joints [48.733, -71.733, 79.61, -0.869, 82.136, 48.849]
  MoveL 458 to (168.35, 120.65, 0) mm, rotated rx -180 ry 0 rz -39.83 deg; joints [48.732, -71.819, 79.723, -0.869, 82.108, 48.848]
  MoveL 459 to (168.37, 119.62, 0) mm, rotated rx 180 ry 0 rz -39.83 deg; joints [48.732, -71.905, 79.837, -0.869, 82.081, 48.849]
  MoveL 460 to (168.4, 118.86, 0) mm, rotated rx 180 ry 0 rz -39.83 deg; joints [48.732, -71.969, 79.921, -0.869, 82.06, 48.849]
  MoveL 461 to (168.44, 118.1, 0) mm, rotated rx -180 ry 0 rz -39.83 deg; joints [48.733, -72.033, 80.005, -0.869, 82.04, 48.851]
  MoveL 462 to (168.49, 117.33, 0) mm, rotated rx 180 ry 0 rz -39.83 deg; joints [48.735, -72.096, 80.089, -0.869, 82.02, 48.853]
  MoveL 463 to (168.55, 116.57, 0) mm, rotated rx 180 ry 0 rz -39.83 deg; joints [48.737, -72.16, 80.173, -0.869, 82, 48.855]
  MoveL 464 to (168.68, 115.28, 0) mm, rotated rx -180 ry 0 rz -39.83 deg; joints [48.742, -72.267, 80.314, -0.869, 81.966, 48.86]
  MoveL 465 to (168.83, 114, 0) mm, rotated rx -180 ry 0 rz -39.83 deg; joints [48.748, -72.375, 80.455, -0.869, 81.932, 48.867]
  MoveL 466 to (169.01, 112.71, 0) mm, rotated rx 180 ry 0 rz -39.83 deg; joints [48.756, -72.482, 80.596, -0.869, 81.898, 48.875]
  MoveL 467 to (169.21, 111.43, 0) mm, rotated rx 180 ry 0 rz -39.83 deg; joints [48.764, -72.589, 80.737, -0.869, 81.865, 48.884]
  MoveL 468 to (169.46, 109.92, 0) mm, rotated rx -180 ry 0 rz -39.83 deg; joints [48.775, -72.715, 80.901, -0.869, 81.826, 48.896]
  MoveL 469 to (169.74, 108.42, 0) mm, rotated rx 180 ry 0 rz -39.83 deg; joints [48.788, -72.84, 81.065, -0.869, 81.788, 48.909]
  MoveL 470 to (170.05, 106.93, 0) mm, rotated rx 180 ry 0 rz -39.83 deg; joints [48.802, -72.964, 81.228, -0.87, 81.75, 48.924]
  MoveL 471 to (170.4, 105.45, 0) mm, rotated rx 180 ry 0 rz -39.83 deg; joints [48.818, -73.088, 81.389, -0.87, 81.713, 48.94]
  MoveL 472 to (170.63, 104.55, 0) mm, rotated rx 180 ry 0 rz -39.83 deg; joints [48.829, -73.163, 81.487, -0.87, 81.69, 48.951]
  MoveL 473 to (170.88, 103.66, 0) mm, rotated rx -180 ry 0 rz -39.83 deg; joints [48.841, -73.237, 81.583, -0.87, 81.668, 48.963]
  MoveL 474 to (171.15, 102.78, 0) mm, rotated rx 180 ry 0 rz -39.83 deg; joints [48.853, -73.311, 81.679, -0.87, 81.646, 48.977]
  MoveL 475 to (171.44, 101.9, 0) mm, rotated rx 180 ry 0 rz -39.83 deg; joints [48.867, -73.384, 81.775, -0.87, 81.624, 48.991]
  MoveL 476 to (171.81, 100.89, 0) mm, rotated rx -180 ry 0 rz -39.83 deg; joints [48.885, -73.469, 81.885, -0.87, 81.599, 49.009]
  MoveL 477 to (172.2, 99.88, 0) mm, rotated rx 180 ry 0 rz -39.83 deg; joints [48.904, -73.553, 81.994, -0.87, 81.574, 49.028]
  MoveL 478 to (172.6, 98.88, 0) mm, rotated rx -180 ry 0 rz -39.83 deg; joints [48.923, -73.636, 82.102, -0.87, 81.549, 49.048]
  MoveL 479 to (173.02, 97.89, 0) mm, rotated rx -180 ry 0 rz -39.83 deg; joints [48.944, -73.719, 82.21, -0.87, 81.525, 49.069]
  MoveL 480 to (173.38, 97.04, 0) mm, rotated rx 180 ry 0 rz -39.83 deg; joints [48.962, -73.79, 82.301, -0.87, 81.505, 49.087]
  MoveL 481 to (173.76, 96.21, 0) mm, rotated rx -180 ry 0 rz -39.83 deg; joints [48.98, -73.859, 82.391, -0.87, 81.484, 49.106]
  MoveL 482 to (174.16, 95.39, 0) mm, rotated rx 180 ry 0 rz -39.83 deg; joints [49, -73.928, 82.48, -0.87, 81.464, 49.126]
  MoveL 483 to (174.6, 94.59, 0) mm, rotated rx 180 ry 0 rz -39.83 deg; joints [49.022, -73.995, 82.566, -0.87, 81.445, 49.148]
  MoveL 484 to (174.88, 94.11, 0) mm, rotated rx 180 ry 0 rz -39.83 deg; joints [49.036, -74.035, 82.618, -0.87, 81.434, 49.163]
  MoveL 485 to (175.19, 93.65, 0) mm, rotated rx 180 ry 0 rz -39.83 deg; joints [49.052, -74.073, 82.668, -0.87, 81.423, 49.179]
  MoveL 486 to (175.51, 93.19, 0) mm, rotated rx 180 ry 0 rz -39.83 deg; joints [49.068, -74.112, 82.717, -0.87, 81.412, 49.195]
  MoveL 487 to (175.85, 92.74, 0) mm, rotated rx -180 ry 0 rz -39.83 deg; joints [49.085, -74.149, 82.766, -0.87, 81.401, 49.212]
  MoveL 488 to (176.14, 92.38, 0) mm, rotated rx -180 ry 0 rz -39.83 deg; joints [49.1, -74.18, 82.806, -0.87, 81.392, 49.227]
  MoveL 489 to (176.44, 92.03, 0) mm, rotated rx 180 ry 0 rz -39.83 deg; joints [49.115, -74.209, 82.844, -0.87, 81.383, 49.243]
  MoveL 490 to (176.77, 91.7, 0) mm, rotated rx 180 ry 0 rz -39.83 deg; joints [49.132, -74.237, 82.88, -0.87, 81.376, 49.259]
  MoveL 491 to (177.13, 91.41, 0) mm, rotated rx 180 ry 0 rz -39.83 deg; joints [49.15, -74.261, 82.912, -0.87, 81.368, 49.278]
  MoveL 492 to (177.41, 91.21, 0) mm, rotated rx 180 ry 0 rz -39.83 deg; joints [49.165, -74.278, 82.933, -0.87, 81.364, 49.293]
  MoveL 493 to (177.72, 91.04, 0) mm, rotated rx 180 ry 0 rz -39.83 deg; joints [49.181, -74.292, 82.952, -0.87, 81.359, 49.308]
  MoveL 494 to (178.03, 90.88, 0) mm, rotated rx -180 ry 0 rz -39.83 deg; joints [49.197, -74.306, 82.97, -0.87, 81.356, 49.324]
  MoveL 495 to (178.34, 90.72, 0) mm, rotated rx 180 ry 0 rz -39.83 deg; joints [49.213, -74.319, 82.987, -0.87, 81.352, 49.341]
  MoveL 496 to (178.56, 90.62, 0) mm, rotated rx 180 ry 0 rz -39.83 deg; joints [49.224, -74.328, 82.999, -0.87, 81.349, 49.352]
  MoveL 497 to (178.78, 90.52, 0) mm, rotated rx 180 ry 0 rz -39.83 deg; joints [49.235, -74.337, 83.01, -0.87, 81.347, 49.363]
  MoveL 498 to (179, 90.43, 0) mm, rotated rx 180 ry 0 rz -39.83 deg; joints [49.247, -74.344, 83.02, -0.87, 81.344, 49.375]
  MoveL 499 to (179.24, 90.37, 0) mm, rotated rx 180 ry 0 rz -39.83 deg; joints [49.259, -74.35, 83.028, -0.87, 81.343, 49.387]
  MoveL 500 to (179.39, 90.34, 0) mm, rotated rx 180 ry 0 rz -39.83 deg; joints [49.267, -74.352, 83.031, -0.87, 81.342, 49.395]
  MoveL 501 to (179.54, 90.33, 0) mm, rotated rx 180 ry 0 rz -39.83 deg; joints [49.275, -74.353, 83.032, -0.87, 81.342, 49.403]
  MoveL 502 to (179.69, 90.34, 0) mm, rotated rx 180 ry 0 rz -39.83 deg; joints [49.283, -74.353, 83.032, -0.87, 81.342, 49.411]
  MoveL 503 to (179.83, 90.37, 0) mm, rotated rx -180 ry 0 rz -39.83 deg; joints [49.29, -74.351, 83.029, -0.87, 81.342, 49.418]
  MoveL 504 to (179.9, 90.39, 0) mm, rotated rx 180 ry 0 rz -39.83 deg; joints [49.294, -74.349, 83.027, -0.87, 81.343, 49.422]
  MoveL 505 to (179.97, 90.42, 0) mm, rotated rx 180 ry 0 rz -39.83 deg; joints [49.297, -74.346, 83.024, -0.87, 81.343, 49.425]
  MoveL 506 to (180.03, 90.45, 0) mm, rotated rx 180 ry 0 rz -39.83 deg; joints [49.301, -74.344, 83.021, -0.87, 81.344, 49.429]
  MoveL 507 to (180.1, 90.49, 0) mm, rotated rx 180 ry 0 rz -39.83 deg; joints [49.304, -74.341, 83.017, -0.87, 81.345, 49.432]
  MoveL 508 to (180.19, 90.54, 0) mm, rotated rx 180 ry 0 rz -39.83 deg; joints [49.309, -74.337, 83.012, -0.87, 81.346, 49.437]
  MoveL 509 to (180.28, 90.59, 0) mm, rotated rx 180 ry 0 rz -39.83 deg; joints [49.314, -74.333, 83.007, -0.87, 81.347, 49.442]
  MoveL 510 to (180.37, 90.64, 0) mm, rotated rx 180 ry 0 rz -39.83 deg; joints [49.318, -74.329, 83.002, -0.87, 81.348, 49.446]
  MoveL 511 to (180.46, 90.69, 0) mm, rotated rx 180 ry 0 rz -39.83 deg; joints [49.323, -74.324, 82.996, -0.87, 81.349, 49.451]
  MoveL 512 to (180.64, 90.83, 0) mm, rotated rx 180 ry 0 rz -39.83 deg; joints [49.333, -74.313, 82.982, -0.87, 81.352, 49.46]
  MoveL 513 to (180.81, 90.99, 0) mm, rotated rx 180 ry 0 rz -39.83 deg; joints [49.342, -74.3, 82.966, -0.87, 81.356, 49.469]
  MoveL 514 to (180.98, 91.15, 0) mm, rotated rx -180 ry 0 rz -39.83 deg; joints [49.35, -74.287, 82.949, -0.87, 81.359, 49.478]
  MoveL 515 to (181.14, 91.32, 0) mm, rotated rx 180 ry 0 rz -39.83 deg; joints [49.359, -74.273, 82.932, -0.87, 81.363, 49.487]
  MoveL 516 to (181.47, 91.67, 0) mm, rotated rx 180 ry 0 rz -39.83 deg; joints [49.376, -74.244, 82.895, -0.87, 81.371, 49.504]
  MoveL 517 to (181.8, 92.02, 0) mm, rotated rx 180 ry 0 rz -39.83 deg; joints [49.394, -74.216, 82.859, -0.87, 81.379, 49.521]
  MoveL 518 to (182.11, 92.38, 0) mm, rotated rx 180 ry 0 rz -39.83 deg; joints [49.41, -74.186, 82.822, -0.87, 81.387, 49.538]
  MoveL 519 to (182.42, 92.74, 0) mm, rotated rx 180 ry 0 rz -39.83 deg; joints [49.426, -74.156, 82.784, -0.87, 81.395, 49.554]
  MoveL 520 to (182.74, 93.14, 0) mm, rotated rx -180 ry 0 rz -39.83 deg; joints [49.443, -74.123, 82.742, -0.87, 81.404, 49.57]
  MoveL 521 to (183.04, 93.55, 0) mm, rotated rx 180 ry 0 rz -39.83 deg; joints [49.459, -74.09, 82.699, -0.87, 81.414, 49.586]
  MoveL 522 to (183.34, 93.97, 0) mm, rotated rx 180 ry 0 rz -39.83 deg; joints [49.475, -74.056, 82.656, -0.87, 81.423, 49.602]
  MoveL 523 to (183.64, 94.38, 0) mm, rotated rx 180 ry 0 rz -39.83 deg; joints [49.491, -74.022, 82.613, -0.87, 81.433, 49.617]
  MoveL 524 to (183.9, 94.74, 0) mm, rotated rx 180 ry 0 rz -39.83 deg; joints [49.505, -73.992, 82.575, -0.87, 81.441, 49.631]
  MoveL 525 to (184.16, 95.1, 0) mm, rotated rx 180 ry 0 rz -39.83 deg; joints [49.518, -73.963, 82.538, -0.87, 81.449, 49.645]
  MoveL 526 to (184.41, 95.46, 0) mm, rotated rx 180 ry 0 rz -39.83 deg; joints [49.532, -73.933, 82.499, -0.87, 81.458, 49.658]
  MoveL 527 to (184.65, 95.84, 0) mm, rotated rx 180 ry 0 rz -39.83 deg; joints [49.544, -73.902, 82.46, -0.87, 81.466, 49.67]
  MoveL 528 to (184.78, 96.05, 0) mm, rotated rx -180 ry 0 rz -39.83 deg; joints [49.551, -73.884, 82.437, -0.87, 81.471, 49.677]
  MoveL 529 to (184.91, 96.27, 0) mm, rotated rx 180 ry 0 rz -39.83 deg; joints [49.558, -73.866, 82.414, -0.87, 81.477, 49.684]
  MoveL 530 to (185.03, 96.5, 0) mm, rotated rx -180 ry 0 rz -39.83 deg; joints [49.564, -73.847, 82.39, -0.87, 81.482, 49.69]
  MoveL 531 to (185.15, 96.72, 0) mm, rotated rx 180 ry 0 rz -39.83 deg; joints [49.571, -73.829, 82.367, -0.87, 81.487, 49.696]
  Establecer velocidad (1000.0 mm/s)
  MoveL 532 to (185.15, 96.72, 0) mm, rotated rx 180 ry 0 rz -39.83 deg; joints [49.571, -73.829, 82.367, -0.87, 81.487, 49.696]
  MoveL 533 to (185.15, 96.72, 20) mm, rotated rx 180 ry 0 rz -39.83 deg; joints [49.586, -74.143, 81.032, -0.867, 83.136, 49.687]
  Establecer velocidad (1000.0 mm/s)
  MoveL 534 to (171.34, 145.91, 20) mm, rotated rx 180 ry 0 rz -39.83 deg; joints [48.927, -69.987, 75.547, -0.865, 84.455, 49.007]
  MoveL 535 to (171.34, 145.91, 0) mm, rotated rx -180 ry 0 rz -39.83 deg; joints [48.912, -69.708, 76.9, -0.867, 82.823, 49.017]
  MoveL 536 to (171.34, 145.91, 0) mm, rotated rx -180 ry 0 rz -39.83 deg; joints [48.912, -69.708, 76.9, -0.867, 82.823, 49.017]
  Establecer velocidad (50.0 mm/s)
  MoveL 537 to (171.39, 146.46, 0) mm, rotated rx 180 ry 0 rz -39.83 deg; joints [48.915, -69.662, 76.837, -0.867, 82.839, 49.02]
  MoveL 538 to (171.44, 147.01, 0) mm, rotated rx -180 ry 0 rz -39.83 deg; joints [48.918, -69.616, 76.775, -0.867, 82.856, 49.023]
  MoveL 539 to (171.49, 147.56, 0) mm, rotated rx -180 ry 0 rz -39.83 deg; joints [48.921, -69.569, 76.712, -0.867, 82.872, 49.025]
  MoveL 540 to (171.51, 148.11, 0) mm, rotated rx 180 ry 0 rz -39.83 deg; joints [48.923, -69.523, 76.649, -0.867, 82.889, 49.027]
  MoveL 541 to (171.53, 149.49, 0) mm, rotated rx 180 ry 0 rz -39.83 deg; joints [48.925, -69.407, 76.491, -0.867, 82.931, 49.029]
  MoveL 542 to (171.45, 150.86, 0) mm, rotated rx -180 ry 0 rz -39.83 deg; joints [48.923, -69.291, 76.333, -0.867, 82.973, 49.026]
  MoveL 543 to (171.32, 152.23, 0) mm, rotated rx 180 ry 0 rz -39.83 deg; joints [48.918, -69.175, 76.174, -0.867, 83.015, 49.02]
  MoveL 544 to (171.13, 153.6, 0) mm, rotated rx 180 ry 0 rz -39.83 deg; joints [48.91, -69.059, 76.016, -0.867, 83.058, 49.011]
  MoveL 545 to (170.92, 154.79, 0) mm, rotated rx 180 ry 0 rz -39.83 deg; joints [48.901, -68.958, 75.877, -0.867, 83.095, 49.002]
  MoveL 546 to (170.69, 155.98, 0) mm, rotated rx 180 ry 0 rz -39.83 deg; joints [48.891, -68.857, 75.739, -0.867, 83.133, 48.991]
  MoveL 547 to (170.41, 157.15, 0) mm, rotated rx 180 ry 0 rz -39.83 deg; joints [48.879, -68.758, 75.602, -0.867, 83.17, 48.978]
  MoveL 548 to (170.09, 158.31, 0) mm, rotated rx 180 ry 0 rz -39.83 deg; joints [48.864, -68.659, 75.466, -0.867, 83.207, 48.963]
  MoveL 549 to (169.78, 159.26, 0) mm, rotated rx 180 ry 0 rz -39.83 deg; joints [48.85, -68.578, 75.355, -0.867, 83.237, 48.949]
  MoveL 550 to (169.44, 160.19, 0) mm, rotated rx 180 ry 0 rz -39.83 deg; joints [48.834, -68.498, 75.244, -0.867, 83.267, 48.933]
  MoveL 551 to (169.07, 161.11, 0) mm, rotated rx 180 ry 0 rz -39.83 deg; joints [48.817, -68.419, 75.135, -0.866, 83.297, 48.915]
  MoveL 552 to (168.66, 162.02, 0) mm, rotated rx -180 ry 0 rz -39.83 deg; joints [48.798, -68.341, 75.027, -0.866, 83.327, 48.896]
  MoveL 553 to (168.32, 162.73, 0) mm, rotated rx -180 ry 0 rz -39.83 deg; joints [48.783, -68.281, 74.943, -0.866, 83.35, 48.88]
  MoveL 554 to (167.96, 163.43, 0) mm, rotated rx -180 ry 0 rz -39.83 deg; joints [48.766, -68.221, 74.86, -0.866, 83.373, 48.863]
  MoveL 555 to (167.58, 164.11, 0) mm, rotated rx -180 ry 0 rz -39.83 deg; joints [48.748, -68.162, 74.778, -0.866, 83.396, 48.845]
  MoveL 556 to (167.18, 164.79, 0) mm, rotated rx 180 ry 0 rz -39.83 deg; joints [48.729, -68.104, 74.697, -0.866, 83.419, 48.826]
  MoveL 557 to (166.6, 165.69, 0) mm, rotated rx 180 ry 0 rz -39.83 deg; joints [48.702, -68.026, 74.588, -0.866, 83.449, 48.798]
  MoveL 558 to (165.99, 166.57, 0) mm, rotated rx 180 ry 0 rz -39.83 deg; joints [48.674, -67.949, 74.482, -0.866, 83.478, 48.769]
  MoveL 559 to (165.35, 167.43, 0) mm, rotated rx 180 ry 0 rz -39.83 deg; joints [48.644, -67.875, 74.378, -0.866, 83.507, 48.738]
  MoveL 560 to (164.67, 168.26, 0) mm, rotated rx 180 ry 0 rz -39.83 deg; joints [48.612, -67.803, 74.277, -0.866, 83.536, 48.706]
  MoveL 561 to (163.97, 169.08, 0) mm, rotated rx 180 ry 0 rz -39.83 deg; joints [48.579, -67.732, 74.178, -0.866, 83.564, 48.673]
  MoveL 562 to (163.25, 169.87, 0) mm, rotated rx 180 ry 0 rz -39.83 deg; joints [48.545, -67.662, 74.08, -0.866, 83.591, 48.638]
  MoveL 563 to (162.5, 170.65, 0) mm, rotated rx 180 ry 0 rz -39.83 deg; joints [48.51, -67.594, 73.985, -0.866, 83.618, 48.603]
  MoveL 564 to (161.74, 171.41, 0) mm, rotated rx -180 ry 0 rz -39.83 deg; joints [48.474, -67.528, 73.891, -0.866, 83.645, 48.567]
  MoveL 565 to (160.92, 172.2, 0) mm, rotated rx 180 ry 0 rz -39.83 deg; joints [48.436, -67.459, 73.794, -0.866, 83.672, 48.528]
  MoveL 566 to (160.09, 172.96, 0) mm, rotated rx 180 ry 0 rz -39.83 deg; joints [48.396, -67.391, 73.699, -0.866, 83.699, 48.488]
  MoveL 567 to (159.23, 173.69, 0) mm, rotated rx 180 ry 0 rz -39.83 deg; joints [48.356, -67.327, 73.608, -0.866, 83.725, 48.447]
  MoveL 568 to (158.33, 174.37, 0) mm, rotated rx 180 ry 0 rz -39.83 deg; joints [48.313, -67.267, 73.523, -0.866, 83.75, 48.404]
  MoveL 569 to (157.25, 175.08, 0) mm, rotated rx 180 ry 0 rz -39.83 deg; joints [48.262, -67.203, 73.432, -0.866, 83.776, 48.353]
  MoveL 570 to (156.13, 175.73, 0) mm, rotated rx -180 ry 0 rz -39.83 deg; joints [48.209, -67.145, 73.349, -0.866, 83.8, 48.3]
  MoveL 571 to (154.97, 176.32, 0) mm, rotated rx 180 ry 0 rz -39.83 deg; joints [48.154, -67.091, 73.273, -0.866, 83.822, 48.244]
  MoveL 572 to (153.79, 176.86, 0) mm, rotated rx 180 ry 0 rz -39.83 deg; joints [48.098, -67.041, 73.202, -0.866, 83.842, 48.188]
  MoveL 573 to (152.22, 177.5, 0) mm, rotated rx 180 ry 0 rz -39.83 deg; joints [48.024, -66.982, 73.116, -0.866, 83.867, 48.113]
  MoveL 574 to (150.63, 178.08, 0) mm, rotated rx -180 ry 0 rz -39.83 deg; joints [47.948, -66.928, 73.038, -0.866, 83.89, 48.037]
  MoveL 575 to (149.02, 178.58, 0) mm, rotated rx 180 ry 0 rz -39.83 deg; joints [47.872, -66.88, 72.969, -0.866, 83.91, 47.96]
  MoveL 576 to (147.38, 178.99, 0) mm, rotated rx 180 ry 0 rz -39.83 deg; joints [47.794, -66.839, 72.909, -0.865, 83.927, 47.882]
  MoveL 577 to (146.39, 179.2, 0) mm, rotated rx 180 ry 0 rz -39.83 deg; joints [47.747, -66.817, 72.878, -0.865, 83.936, 47.835]
  MoveL 578 to (145.4, 179.38, 0) mm, rotated rx 180 ry 0 rz -39.83 deg; joints [47.699, -66.798, 72.85, -0.865, 83.945, 47.787]
  MoveL 579 to (144.39, 179.53, 0) mm, rotated rx 180 ry 0 rz -39.83 deg; joints [47.651, -66.782, 72.826, -0.865, 83.952, 47.739]
  MoveL 580 to (143.39, 179.64, 0) mm, rotated rx 180 ry 0 rz -39.83 deg; joints [47.603, -66.769, 72.806, -0.865, 83.958, 47.691]
  MoveL 581 to (141.57, 179.76, 0) mm, rotated rx -180 ry 0 rz -39.83 deg; joints [47.516, -66.752, 72.781, -0.865, 83.965, 47.604]
  MoveL 582 to (139.74, 179.75, 0) mm, rotated rx 180 ry 0 rz -39.83 deg; joints [47.428, -66.746, 72.769, -0.865, 83.969, 47.516]
  MoveL 583 to (137.93, 179.62, 0) mm, rotated rx -180 ry 0 rz -39.83 deg; joints [47.341, -66.75, 72.772, -0.865, 83.969, 47.428]
  MoveL 584 to (136.13, 179.35, 0) mm, rotated rx -180 ry 0 rz -39.83 deg; joints [47.254, -66.766, 72.792, -0.865, 83.963, 47.342]
  MoveL 585 to (135.08, 179.12, 0) mm, rotated rx 180 ry 0 rz -39.83 deg; joints [47.203, -66.781, 72.812, -0.865, 83.958, 47.29]
  MoveL 586 to (134.03, 178.85, 0) mm, rotated rx -180 ry 0 rz -39.83 deg; joints [47.152, -66.8, 72.837, -0.865, 83.951, 47.24]
  MoveL 587 to (133, 178.55, 0) mm, rotated rx 180 ry 0 rz -39.83 deg; joints [47.101, -66.82, 72.865, -0.865, 83.943, 47.189]
  MoveL 588 to (131.96, 178.24, 0) mm, rotated rx 180 ry 0 rz -39.83 deg; joints [47.051, -66.842, 72.895, -0.865, 83.935, 47.139]
  MoveL 589 to (131.96, 178.24, 0) mm, rotated rx 180 ry 0 rz -39.83 deg; joints [47.051, -66.842, 72.895, -0.865, 83.935, 47.139]
  MoveL 590 to (131.9, 178.2, 0) mm, rotated rx 180 ry 0 rz -39.83 deg; joints [47.048, -66.845, 72.899, -0.865, 83.933, 47.136]
  MoveL 591 to (131.85, 178.16, 0) mm, rotated rx 180 ry 0 rz -39.83 deg; joints [47.045, -66.849, 72.903, -0.865, 83.932, 47.133]
  MoveL 592 to (131.81, 178.12, 0) mm, rotated rx 180 ry 0 rz -39.83 deg; joints [47.043, -66.852, 72.908, -0.865, 83.931, 47.131]
  MoveL 593 to (131.77, 178.07, 0) mm, rotated rx 180 ry 0 rz -39.83 deg; joints [47.041, -66.856, 72.914, -0.865, 83.929, 47.129]
  MoveL 594 to (131.74, 177.98, 0) mm, rotated rx 180 ry 0 rz -39.83 deg; joints [47.039, -66.864, 72.925, -0.865, 83.926, 47.128]
  MoveL 595 to (131.74, 177.87, 0) mm, rotated rx -180 ry 0 rz -39.83 deg; joints [47.039, -66.874, 72.938, -0.865, 83.922, 47.127]
  MoveL 596 to (131.75, 177.75, 0) mm, rotated rx 180 ry 0 rz -39.83 deg; joints [47.039, -66.884, 72.952, -0.865, 83.918, 47.128]
  MoveL 597 to (131.78, 177.63, 0) mm, rotated rx -180 ry 0 rz -39.83 deg; joints [47.04, -66.894, 72.966, -0.865, 83.914, 47.129]
  MoveL 598 to (131.8, 177.5, 0) mm, rotated rx -180 ry 0 rz -39.83 deg; joints [47.041, -66.905, 72.983, -0.865, 83.909, 47.13]
  MoveL 599 to (131.83, 177.37, 0) mm, rotated rx -180 ry 0 rz -39.83 deg; joints [47.042, -66.917, 72.998, -0.865, 83.905, 47.131]
  MoveL 600 to (131.86, 177.25, 0) mm, rotated rx -180 ry 0 rz -39.83 deg; joints [47.043, -66.927, 73.014, -0.865, 83.9, 47.132]
  MoveL 601 to (131.9, 177.12, 0) mm, rotated rx -180 ry 0 rz -39.83 deg; joints [47.044, -66.938, 73.029, -0.865, 83.896, 47.133]
  MoveL 602 to (131.96, 176.92, 0) mm, rotated rx -180 ry 0 rz -39.83 deg; joints [47.047, -66.956, 73.054, -0.865, 83.889, 47.136]
  MoveL 603 to (132.04, 176.72, 0) mm, rotated rx 180 ry 0 rz -39.83 deg; joints [47.05, -66.973, 73.078, -0.865, 83.882, 47.139]
  MoveL 604 to (132.13, 176.52, 0) mm, rotated rx 180 ry 0 rz -39.83 deg; joints [47.054, -66.991, 73.103, -0.865, 83.875, 47.143]
  MoveL 605 to (132.22, 176.32, 0) mm, rotated rx 180 ry 0 rz -39.83 deg; joints [47.058, -67.008, 73.127, -0.865, 83.868, 47.147]
  MoveL 606 to (132.38, 176.01, 0) mm, rotated rx 180 ry 0 rz -39.83 deg; joints [47.065, -67.036, 73.166, -0.865, 83.857, 47.154]
  MoveL 607 to (132.55, 175.7, 0) mm, rotated rx 180 ry 0 rz -39.83 deg; joints [47.072, -67.063, 73.204, -0.866, 83.846, 47.162]
  MoveL 608 to (132.73, 175.4, 0) mm, rotated rx 180 ry 0 rz -39.83 deg; joints [47.08, -67.089, 73.242, -0.866, 83.835, 47.17]
  MoveL 609 to (132.92, 175.1, 0) mm, rotated rx -180 ry 0 rz -39.83 deg; joints [47.089, -67.115, 73.278, -0.866, 83.825, 47.178]
  MoveL 610 to (133.39, 174.43, 0) mm, rotated rx 180 ry 0 rz -39.83 deg; joints [47.11, -67.175, 73.362, -0.866, 83.8, 47.2]
  MoveL 611 to (133.9, 173.78, 0) mm, rotated rx 180 ry 0 rz -39.83 deg; joints [47.132, -67.233, 73.444, -0.866, 83.777, 47.223]
  MoveL 612 to (134.43, 173.14, 0) mm, rotated rx 180 ry 0 rz -39.83 deg; joints [47.156, -67.289, 73.523, -0.866, 83.754, 47.247]
  MoveL 613 to (134.97, 172.52, 0) mm, rotated rx 180 ry 0 rz -39.83 deg; joints [47.181, -67.345, 73.602, -0.866, 83.732, 47.272]
  MoveL 614 to (136.32, 170.96, 0) mm, rotated rx 180 ry 0 rz -39.83 deg; joints [47.242, -67.484, 73.797, -0.866, 83.677, 47.334]
  MoveL 615 to (137.7, 169.43, 0) mm, rotated rx 180 ry 0 rz -39.83 deg; joints [47.305, -67.62, 73.988, -0.866, 83.623, 47.398]
  MoveL 616 to (139.1, 167.93, 0) mm, rotated rx -180 ry 0 rz -39.83 deg; joints [47.369, -67.754, 74.176, -0.866, 83.57, 47.463]
  MoveL 617 to (140.54, 166.46, 0) mm, rotated rx 180 ry 0 rz -39.83 deg; joints [47.436, -67.884, 74.358, -0.866, 83.518, 47.53]
  MoveL 618 to (142.13, 164.94, 0) mm, rotated rx 180 ry 0 rz -39.83 deg; joints [47.51, -68.02, 74.548, -0.866, 83.465, 47.605]
  MoveL 619 to (143.76, 163.45, 0) mm, rotated rx 180 ry 0 rz -39.83 deg; joints [47.586, -68.152, 74.734, -0.866, 83.413, 47.682]
  MoveL 620 to (145.42, 161.99, 0) mm, rotated rx 180 ry 0 rz -39.83 deg; joints [47.664, -68.282, 74.916, -0.866, 83.363, 47.761]
  MoveL 621 to (147.09, 160.53, 0) mm, rotated rx -180 ry 0 rz -39.83 deg; joints [47.742, -68.412, 75.096, -0.867, 83.313, 47.84]
  MoveL 622 to (149.36, 158.54, 0) mm, rotated rx 180 ry 0 rz -39.83 deg; joints [47.849, -68.588, 75.342, -0.867, 83.245, 47.948]
  MoveL 623 to (151.65, 156.58, 0) mm, rotated rx -180 ry 0 rz -39.83 deg; joints [47.957, -68.761, 75.582, -0.867, 83.179, 48.057]
  MoveL 624 to (153.99, 154.69, 0) mm, rotated rx 180 ry 0 rz -39.83 deg; joints [48.069, -68.928, 75.815, -0.867, 83.116, 48.169]
  MoveL 625 to (156.4, 152.9, 0) mm, rotated rx 180 ry 0 rz -39.83 deg; joints [48.184, -69.086, 76.034, -0.867, 83.056, 48.286]
  MoveL 626 to (158.01, 151.81, 0) mm, rotated rx -180 ry 0 rz -39.83 deg; joints [48.261, -69.182, 76.167, -0.867, 83.02, 48.364]
  MoveL 627 to (159.64, 150.76, 0) mm, rotated rx -180 ry 0 rz -39.83 deg; joints [48.34, -69.275, 76.296, -0.867, 82.985, 48.443]
  MoveL 628 to (161.29, 149.72, 0) mm, rotated rx 180 ry 0 rz -39.83 deg; joints [48.42, -69.367, 76.423, -0.867, 82.951, 48.523]
  MoveL 629 to (162.93, 148.68, 0) mm, rotated rx 180 ry 0 rz -39.83 deg; joints [48.5, -69.459, 76.55, -0.867, 82.917, 48.603]
  MoveL 630 to (163.98, 148, 0) mm, rotated rx 180 ry 0 rz -39.83 deg; joints [48.55, -69.518, 76.633, -0.867, 82.895, 48.654]
  MoveL 631 to (165.03, 147.34, 0) mm, rotated rx 180 ry 0 rz -39.83 deg; joints [48.601, -69.576, 76.713, -0.867, 82.874, 48.706]
  MoveL 632 to (166.1, 146.72, 0) mm, rotated rx 180 ry 0 rz -39.83 deg; joints [48.653, -69.63, 76.788, -0.867, 82.854, 48.758]
  MoveL 633 to (167.22, 146.19, 0) mm, rotated rx 180 ry 0 rz -39.83 deg; joints [48.708, -69.678, 76.854, -0.867, 82.836, 48.813]
  MoveL 634 to (167.63, 146.01, 0) mm, rotated rx 180 ry 0 rz -39.83 deg; joints [48.728, -69.693, 76.875, -0.867, 82.83, 48.834]
  MoveL 635 to (168.06, 145.86, 0) mm, rotated rx 180 ry 0 rz -39.83 deg; joints [48.749, -69.707, 76.894, -0.867, 82.825, 48.855]
  MoveL 636 to (168.49, 145.71, 0) mm, rotated rx 180 ry 0 rz -39.83 deg; joints [48.77, -69.72, 76.913, -0.867, 82.82, 48.876]
  MoveL 637 to (168.91, 145.57, 0) mm, rotated rx 180 ry 0 rz -39.83 deg; joints [48.791, -69.732, 76.93, -0.867, 82.815, 48.897]
  MoveL 638 to (169.24, 145.48, 0) mm, rotated rx 180 ry 0 rz -39.83 deg; joints [48.807, -69.741, 76.942, -0.867, 82.812, 48.913]
  MoveL 639 to (169.57, 145.4, 0) mm, rotated rx 180 ry 0 rz -39.83 deg; joints [48.824, -69.748, 76.952, -0.867, 82.809, 48.929]
  MoveL 640 to (169.91, 145.34, 0) mm, rotated rx 180 ry 0 rz -39.83 deg; joints [48.84, -69.754, 76.96, -0.867, 82.807, 48.946]
  MoveL 641 to (170.26, 145.32, 0) mm, rotated rx 180 ry 0 rz -39.83 deg; joints [48.858, -69.756, 76.964, -0.867, 82.806, 48.963]
  MoveL 642 to (170.47, 145.33, 0) mm, rotated rx 180 ry 0 rz -39.83 deg; joints [48.868, -69.756, 76.964, -0.867, 82.806, 48.974]
  MoveL 643 to (170.69, 145.36, 0) mm, rotated rx -180 ry 0 rz -39.83 deg; joints [48.879, -69.754, 76.961, -0.867, 82.807, 48.984]
  MoveL 644 to (170.88, 145.42, 0) mm, rotated rx 180 ry 0 rz -39.83 deg; joints [48.889, -69.749, 76.955, -0.867, 82.809, 48.994]
  MoveL 645 to (171.05, 145.52, 0) mm, rotated rx 180 ry 0 rz -39.83 deg; joints [48.897, -69.74, 76.944, -0.867, 82.811, 49.003]
  MoveL 646 to (171.14, 145.61, 0) mm, rotated rx 180 ry 0 rz -39.83 deg; joints [48.902, -69.734, 76.934, -0.867, 82.814, 49.007]
  MoveL 647 to (171.21, 145.7, 0) mm, rotated rx -180 ry 0 rz -39.83 deg; joints [48.905, -69.726, 76.924, -0.867, 82.817, 49.011]
  MoveL 648 to (171.28, 145.8, 0) mm, rotated rx -180 ry 0 rz -39.83 deg; joints [48.909, -69.717, 76.912, -0.867, 82.82, 49.014]
  MoveL 649 to (171.34, 145.91, 0) mm, rotated rx -180 ry 0 rz -39.83 deg; joints [48.912, -69.708, 76.9, -0.867, 82.823, 49.017]
  Establecer velocidad (1000.0 mm/s)
  MoveL 650 to (171.34, 145.91, 0) mm, rotated rx -180 ry 0 rz -39.83 deg; joints [48.912, -69.708, 76.9, -0.867, 82.823, 49.017]
  MoveL 651 to (171.34, 145.91, 20) mm, rotated rx 180 ry 0 rz -39.83 deg; joints [48.927, -69.987, 75.547, -0.865, 84.455, 49.007]
  Establecer velocidad (1000.0 mm/s)
  MoveL 652 to (101.69, 155.36, 20) mm, rotated rx 180 ry 0 rz -39.83 deg; joints [45.523, -68.888, 73.963, -0.863, 84.889, 45.597]
  MoveL 653 to (101.69, 155.36, 0) mm, rotated rx 180 ry 0 rz -39.83 deg; joints [45.508, -68.621, 75.325, -0.866, 83.26, 45.607]
  MoveL 654 to (101.69, 155.36, 0) mm, rotated rx 180 ry 0 rz -39.83 deg; joints [45.508, -68.621, 75.325, -0.866, 83.26, 45.607]
  Establecer velocidad (50.0 mm/s)
  MoveL 655 to (102.25, 155.37, 0) mm, rotated rx 180 ry 0 rz -39.83 deg; joints [45.536, -68.624, 75.33, -0.866, 83.258, 45.634]
  MoveL 656 to (102.81, 155.38, 0) mm, rotated rx 180 ry 0 rz -39.83 deg; joints [45.563, -68.627, 75.334, -0.866, 83.257, 45.661]
  MoveL 657 to (103.36, 155.4, 0) mm, rotated rx 180 ry 0 rz -39.83 deg; joints [45.59, -68.629, 75.338, -0.866, 83.256, 45.688]
  MoveL 658 to (103.92, 155.42, 0) mm, rotated rx -180 ry 0 rz -39.83 deg; joints [45.617, -68.63, 75.341, -0.866, 83.255, 45.716]
  MoveL 659 to (104.95, 155.49, 0) mm, rotated rx -180 ry 0 rz -39.83 deg; joints [45.668, -68.631, 75.343, -0.866, 83.254, 45.766]
  MoveL 660 to (105.98, 155.59, 0) mm, rotated rx 180 ry 0 rz -39.83 deg; joints [45.719, -68.63, 75.342, -0.866, 83.254, 45.817]
  MoveL 661 to (107.01, 155.71, 0) mm, rotated rx 180 ry 0 rz -39.83 deg; joints [45.77, -68.626, 75.339, -0.866, 83.255, 45.868]
  MoveL 662 to (108.04, 155.86, 0) mm, rotated rx 180 ry 0 rz -39.83 deg; joints [45.82, -68.62, 75.332, -0.866, 83.256, 45.918]
  MoveL 663 to (108.88, 155.99, 0) mm, rotated rx -180 ry 0 rz -39.83 deg; joints [45.862, -68.614, 75.325, -0.866, 83.258, 45.96]
  MoveL 664 to (109.73, 156.14, 0) mm, rotated rx 180 ry 0 rz -39.83 deg; joints [45.904, -68.606, 75.316, -0.866, 83.261, 46.002]
  MoveL 665 to (110.56, 156.31, 0) mm, rotated rx 180 ry 0 rz -39.83 deg; joints [45.945, -68.597, 75.304, -0.866, 83.263, 46.043]
  MoveL 666 to (111.4, 156.5, 0) mm, rotated rx -180 ry 0 rz -39.83 deg; joints [45.987, -68.586, 75.29, -0.866, 83.267, 46.085]
  MoveL 667 to (112.19, 156.7, 0) mm, rotated rx 180 ry 0 rz -39.83 deg; joints [46.026, -68.574, 75.274, -0.866, 83.271, 46.124]
  MoveL 668 to (112.99, 156.92, 0) mm, rotated rx -180 ry 0 rz -39.83 deg; joints [46.066, -68.56, 75.256, -0.866, 83.276, 46.164]
  MoveL 669 to (113.77, 157.16, 0) mm, rotated rx 180 ry 0 rz -39.83 deg; joints [46.105, -68.544, 75.235, -0.866, 83.282, 46.203]
  MoveL 670 to (114.56, 157.41, 0) mm, rotated rx 180 ry 0 rz -39.83 deg; joints [46.144, -68.528, 75.213, -0.866, 83.287, 46.242]
  MoveL 671 to (115.4, 157.69, 0) mm, rotated rx 180 ry 0 rz -39.83 deg; joints [46.186, -68.508, 75.188, -0.866, 83.294, 46.284]
  MoveL 672 to (116.24, 157.99, 0) mm, rotated rx -180 ry 0 rz -39.83 deg; joints [46.229, -68.488, 75.161, -0.866, 83.302, 46.326]
  MoveL 673 to (117.08, 158.32, 0) mm, rotated rx -180 ry 0 rz -39.83 deg; joints [46.27, -68.465, 75.131, -0.866, 83.31, 46.368]
  MoveL 674 to (117.9, 158.67, 0) mm, rotated rx 180 ry 0 rz -39.83 deg; joints [46.311, -68.44, 75.097, -0.866, 83.319, 46.409]
  MoveL 675 to (118.5, 158.95, 0) mm, rotated rx 180 ry 0 rz -39.83 deg; joints [46.342, -68.419, 75.069, -0.866, 83.326, 46.439]
  MoveL 676 to (119.1, 159.25, 0) mm, rotated rx 180 ry 0 rz -39.83 deg; joints [46.372, -68.397, 75.039, -0.866, 83.334, 46.469]
  MoveL 677 to (119.69, 159.57, 0) mm, rotated rx 180 ry 0 rz -39.83 deg; joints [46.402, -68.374, 75.008, -0.866, 83.343, 46.499]
  MoveL 678 to (120.27, 159.89, 0) mm, rotated rx 180 ry 0 rz -39.83 deg; joints [46.431, -68.349, 74.975, -0.866, 83.352, 46.528]
  MoveL 679 to (120.96, 160.29, 0) mm, rotated rx 180 ry 0 rz -39.83 deg; joints [46.466, -68.318, 74.934, -0.866, 83.363, 46.563]
  MoveL 680 to (121.63, 160.71, 0) mm, rotated rx 180 ry 0 rz -39.83 deg; joints [46.5, -68.286, 74.89, -0.866, 83.375, 46.597]
  MoveL 681 to (122.3, 161.15, 0) mm, rotated rx 180 ry 0 rz -39.83 deg; joints [46.534, -68.253, 74.844, -0.866, 83.387, 46.63]
  MoveL 682 to (122.94, 161.62, 0) mm, rotated rx -180 ry 0 rz -39.83 deg; joints [46.567, -68.216, 74.795, -0.866, 83.401, 46.663]
  MoveL 683 to (123.44, 162.01, 0) mm, rotated rx 180 ry 0 rz -39.83 deg; joints [46.592, -68.186, 74.754, -0.866, 83.412, 46.688]
  MoveL 684 to (123.92, 162.42, 0) mm, rotated rx -180 ry 0 rz -39.83 deg; joints [46.617, -68.154, 74.71, -0.866, 83.424, 46.713]
  MoveL 685 to (124.38, 162.85, 0) mm, rotated rx 180 ry 0 rz -39.83 deg; joints [46.641, -68.119, 74.663, -0.866, 83.437, 46.736]
  MoveL 686 to (124.82, 163.3, 0) mm, rotated rx 180 ry 0 rz -39.83 deg; joints [46.663, -68.083, 74.613, -0.866, 83.451, 46.759]
  MoveL 687 to (125.19, 163.73, 0) mm, rotated rx 180 ry 0 rz -39.83 deg; joints [46.682, -68.048, 74.566, -0.866, 83.464, 46.778]
  MoveL 688 to (125.53, 164.18, 0) mm, rotated rx 180 ry 0 rz -39.83 deg; joints [46.701, -68.012, 74.517, -0.866, 83.477, 46.796]
  MoveL 689 to (125.86, 164.64, 0) mm, rotated rx 180 ry 0 rz -39.83 deg; joints [46.718, -67.975, 74.465, -0.866, 83.492, 46.813]
  MoveL 690 to (126.16, 165.11, 0) mm, rotated rx 180 ry 0 rz -39.83 deg; joints [46.734, -67.936, 74.412, -0.866, 83.506, 46.829]
  MoveL 691 to (126.41, 165.53, 0) mm, rotated rx 180 ry 0 rz -39.83 deg; joints [46.747, -67.902, 74.364, -0.866, 83.519, 46.842]
  MoveL 692 to (126.65, 165.96, 0) mm, rotated rx 180 ry 0 rz -39.83 deg; joints [46.76, -67.866, 74.316, -0.866, 83.533, 46.854]
  MoveL 693 to (126.85, 166.39, 0) mm, rotated rx -180 ry 0 rz -39.83 deg; joints [46.771, -67.83, 74.266, -0.866, 83.547, 46.865]
  MoveL 694 to (127.02, 166.84, 0) mm, rotated rx -180 ry 0 rz -39.83 deg; joints [46.781, -67.793, 74.215, -0.866, 83.561, 46.874]
  MoveL 695 to (127.13, 167.21, 0) mm, rotated rx -180 ry 0 rz -39.83 deg; joints [46.787, -67.762, 74.172, -0.866, 83.573, 46.881]
  MoveL 696 to (127.22, 167.59, 0) mm, rotated rx 180 ry 0 rz -39.83 deg; joints [46.792, -67.73, 74.128, -0.866, 83.585, 46.886]
  MoveL 697 to (127.28, 167.98, 0) mm, rotated rx 180 ry 0 rz -39.83 deg; joints [46.796, -67.698, 74.082, -0.866, 83.598, 46.89]
  MoveL 698 to (127.32, 168.37, 0) mm, rotated rx 180 ry 0 rz -39.83 deg; joints [46.8, -67.664, 74.036, -0.866, 83.611, 46.893]
  MoveL 699 to (127.34, 168.78, 0) mm, rotated rx 180 ry 0 rz -39.83 deg; joints [46.802, -67.63, 73.988, -0.866, 83.625, 46.894]
  MoveL 700 to (127.34, 169.18, 0) mm, rotated rx -180 ry 0 rz -39.83 deg; joints [46.803, -67.595, 73.94, -0.866, 83.638, 46.895]
  MoveL 701 to (127.33, 169.58, 0) mm, rotated rx -180 ry 0 rz -39.83 deg; joints [46.803, -67.561, 73.893, -0.866, 83.651, 46.896]
  MoveL 702 to (127.3, 169.97, 0) mm, rotated rx 180 ry 0 rz -39.83 deg; joints [46.803, -67.528, 73.847, -0.866, 83.664, 46.896]
  MoveL 703 to (127.28, 170.29, 0) mm, rotated rx 180 ry 0 rz -39.83 deg; joints [46.803, -67.5, 73.808, -0.866, 83.675, 46.895]
  MoveL 704 to (127.24, 170.61, 0) mm, rotated rx 180 ry 0 rz -39.83 deg; joints [46.802, -67.473, 73.771, -0.866, 83.686, 46.894]
  MoveL 705 to (127.19, 170.92, 0) mm, rotated rx -180 ry 0 rz -39.83 deg; joints [46.801, -67.446, 73.733, -0.866, 83.697, 46.892]
  MoveL 706 to (127.13, 171.24, 0) mm, rotated rx -180 ry 0 rz -39.83 deg; joints [46.798, -67.419, 73.695, -0.866, 83.707, 46.89]
  MoveL 707 to (127.02, 171.66, 0) mm, rotated rx -180 ry 0 rz -39.83 deg; joints [46.795, -67.382, 73.644, -0.866, 83.722, 46.886]
  MoveL 708 to (126.89, 172.09, 0) mm, rotated rx 180 ry 0 rz -39.83 deg; joints [46.79, -67.345, 73.591, -0.866, 83.737, 46.881]
  MoveL 709 to (126.74, 172.52, 0) mm, rotated rx 180 ry 0 rz -39.83 deg; joints [46.783, -67.308, 73.539, -0.866, 83.752, 46.874]
  MoveL 710 to (126.56, 172.93, 0) mm, rotated rx 180 ry 0 rz -39.83 deg; joints [46.776, -67.272, 73.488, -0.866, 83.766, 46.866]
  MoveL 711 to (126.3, 173.42, 0) mm, rotated rx 180 ry 0 rz -39.83 deg; joints [46.765, -67.229, 73.428, -0.866, 83.783, 46.855]
  MoveL 712 to (126.01, 173.88, 0) mm, rotated rx 180 ry 0 rz -39.83 deg; joints [46.752, -67.188, 73.371, -0.865, 83.799, 46.842]
  MoveL 713 to (125.7, 174.31, 0) mm, rotated rx 180 ry 0 rz -39.83 deg; joints [46.738, -67.149, 73.316, -0.865, 83.815, 46.828]
  MoveL 714 to (125.37, 174.73, 0) mm, rotated rx 180 ry 0 rz -39.83 deg; joints [46.723, -67.112, 73.263, -0.865, 83.83, 46.813]
  MoveL 715 to (124.68, 175.53, 0) mm, rotated rx -180 ry 0 rz -39.83 deg; joints [46.693, -67.04, 73.162, -0.865, 83.859, 46.782]
  MoveL 716 to (123.94, 176.29, 0) mm, rotated rx 180 ry 0 rz -39.83 deg; joints [46.659, -66.971, 73.065, -0.865, 83.887, 46.748]
  MoveL 717 to (123.16, 177.02, 0) mm, rotated rx -180 ry 0 rz -39.83 deg; joints [46.624, -66.905, 72.971, -0.865, 83.914, 46.712]
  MoveL 718 to (122.34, 177.71, 0) mm, rotated rx 180 ry 0 rz -39.83 deg; joints [46.587, -66.842, 72.881, -0.865, 83.94, 46.675]
  MoveL 719 to (121.67, 178.23, 0) mm, rotated rx -180 ry 0 rz -39.83 deg; joints [46.556, -66.794, 72.813, -0.865, 83.96, 46.644]
  MoveL 720 to (120.99, 178.72, 0) mm, rotated rx -180 ry 0 rz -39.83 deg; joints [46.525, -66.748, 72.748, -0.865, 83.979, 46.612]
  MoveL 721 to (120.29, 179.21, 0) mm, rotated rx 180 ry 0 rz -39.83 deg; joints [46.493, -66.703, 72.683, -0.865, 83.998, 46.58]
  MoveL 722 to (119.58, 179.68, 0) mm, rotated rx 180 ry 0 rz -39.83 deg; joints [46.46, -66.659, 72.621, -0.865, 84.016, 46.547]
  MoveL 723 to (118.76, 180.2, 0) mm, rotated rx 180 ry 0 rz -39.83 deg; joints [46.422, -66.609, 72.55, -0.865, 84.037, 46.509]
  MoveL 724 to (117.93, 180.71, 0) mm, rotated rx 180 ry 0 rz -39.83 deg; joints [46.384, -66.561, 72.481, -0.865, 84.057, 46.47]
  MoveL 725 to (117.08, 181.19, 0) mm, rotated rx 180 ry 0 rz -39.83 deg; joints [46.345, -66.515, 72.415, -0.865, 84.076, 46.431]
  MoveL 726 to (116.23, 181.64, 0) mm, rotated rx 180 ry 0 rz -39.83 deg; joints [46.306, -66.472, 72.353, -0.865, 84.094, 46.391]
  MoveL 727 to (115.37, 182.04, 0) mm, rotated rx 180 ry 0 rz -39.83 deg; joints [46.266, -66.433, 72.297, -0.865, 84.111, 46.352]
